C09089=1078.091,60.474,-64.485,173.827,22.395,153.881
C09090=1078.085,60.225,-64.469,173.826,22.393,153.880
C09091=1078.079,59.976,-64.451,173.824,22.391,153.880
C09092=1078.073,59.726,-64.435,173.822,22.388,153.880
C09093=1078.067,59.477,-64.419,173.821,22.386,153.880
C09094=1078.061,59.228,-64.403,173.820,22.383,153.879
C09095=1078.056,58.978,-64.386,173.818,22.381,153.879
C09096=1078.050,58.729,-64.369,173.816,22.379,153.879
C09097=1078.044,58.480,-64.352,173.815,22.376,153.879
C09098=1078.038,58.230,-64.336,173.814,22.374,153.878
C09099=1078.033,57.981,-64.319,173.812,22.371,153.878
C09100=1078.027,57.731,-64.303,173.810,22.369,153.878
C09101=1078.021,57.482,-64.287,173.809,22.367,153.878
C09102=1078.015,57.233,-64.271,173.807,22.364,153.877
C09103=1078.010,56.983,-64.254,173.806,22.362,153.877
C09104=1078.004,56.734,-64.237,173.804,22.359,153.877
C09105=1077.998,56.484,-64.221,173.803,22.357,153.877
C09106=1077.992,56.235,-64.205,173.801,22.354,153.876
C09107=1077.986,55.986,-64.189,173.800,22.352,153.876
C09108=1077.981,55.736,-64.172,173.798,22.350,153.876
C09109=1077.975,55.487,-64.156,173.796,22.347,153.876
C09110=1077.969,55.237,-64.139,173.795,22.344,153.875
C09111=1077.963,54.988,-64.123,173.794,22.342,153.875
C09112=1077.957,54.739,-64.107,173.793,22.340,153.875
C09113=1077.952,54.489,-64.090,173.790,22.337,153.875
C09114=1077.946,54.240,-64.074,173.789,22.335,153.874
C09115=1077.940,53.990,-64.057,173.788,22.332,153.874
C09116=1077.934,53.741,-64.041,173.787,22.330,153.874
C09117=1077.928,53.492,-64.025,173.785,22.328,153.874
C09118=1077.923,53.242,-64.008,173.783,22.325,153.873
C09119=1077.917,52.993,-63.992,173.782,22.323,153.873
C09120=1077.911,52.743,-63.976,173.780,22.320,153.873
C09121=1077.905,52.494,-63.959,173.779,22.317,153.872
C09122=1077.899,52.245,-63.943,173.777,22.316,153.872
C09123=1077.893,51.995,-63.927,173.776,22.313,153.872
C09124=1077.887,51.746,-63.911,173.774,22.310,153.872
C09125=1077.882,51.496,-63.894,173.773,22.308,153.871
C09126=1077.876,51.246,-63.878,173.772,22.305,153.871
C09127=1077.871,50.998,-63.862,173.770,22.303,153.871
C09128=1077.865,50.748,-63.846,173.768,22.301,153.871
C09129=1077.859,50.499,-63.830,173.767,22.298,153.870
C09130=1077.853,50.250,-63.814,173.766,22.296,153.870
C09131=1077.847,50.000,-63.797,173.764,22.293,153.870
C09132=1077.842,49.751,-63.780,173.762,22.290,153.870
C09133=1077.836,49.501,-63.765,173.761,22.288,153.869
C09134=1077.830,49.251,-63.749,173.760,22.286,153.869
C09135=1077.824,49.002,-63.732,173.758,22.283,153.869
C09136=1077.819,48.753,-63.716,173.757,22.281,153.869
C09137=1077.813,48.504,-63.700,173.755,22.278,153.868
C09138=1077.807,48.254,-63.685,173.754,22.276,153.868
C09139=1077.801,48.005,-63.668,173.752,22.273,153.868
C09140=1077.796,47.755,-63.652,173.751,22.271,153.867
C09141=1077.790,47.506,-63.635,173.750,22.268,153.867
C09142=1077.783,47.225,-63.618,173.747,22.265,153.867
C09143=1077.777,46.944,-63.600,173.746,22.263,153.867
C09144=1077.771,46.663,-63.581,173.744,22.260,153.866
C09145=1077.764,46.383,-63.563,173.743,22.257,153.866
C09146=1077.758,46.133,-63.548,173.741,22.254,153.866
C09147=1077.753,45.883,-63.531,173.740,22.252,153.865
C09148=1077.748,45.635,-63.515,173.738,22.250,153.865
C09149=1077.742,45.385,-63.499,173.737,22.247,153.865
C09150=1077.736,45.135,-63.483,173.735,22.244,153.865
C09151=1077.730,44.886,-63.467,173.734,22.242,153.864
C09152=1077.724,44.637,-63.451,173.733,22.240,153.864
C09153=1077.719,44.387,-63.436,173.732,22.237,153.864
C09154=1077.713,44.138,-63.419,173.729,22.234,153.863
C09155=1077.707,43.889,-63.403,173.728,22.232,153.863
C09156=1077.702,43.639,-63.388,173.727,22.229,153.863
C09157=1077.696,43.389,-63.371,173.726,22.227,153.863
C09158=1077.691,43.140,-63.356,173.724,22.225,153.862
C09159=1077.685,42.891,-63.340,173.722,22.222,153.862
C09160=1077.679,42.641,-63.324,173.721,22.220,153.862
C09161=1077.672,42.392,-63.309,173.720,22.217,153.862
C09162=1077.666,42.142,-63.292,173.718,22.215,153.861
C09163=1077.661,41.893,-63.277,173.716,22.212,153.861
C09164=1077.655,41.644,-63.261,173.715,22.210,153.861
C09165=1077.650,41.394,-63.245,173.714,22.208,153.861
C09166=1077.644,41.144,-63.229,173.712,22.205,153.860
C09167=1077.638,40.895,-63.213,173.711,22.202,153.860
C09168=1077.633,40.646,-63.198,173.709,22.200,153.860
C09169=1077.626,40.397,-63.182,173.708,22.198,153.860
C09170=1077.621,40.147,-63.167,173.706,22.195,153.859
C09171=1077.615,39.897,-63.150,173.705,22.193,153.859
C09172=1077.609,39.647,-63.135,173.704,22.190,153.859
C09173=1077.604,39.399,-63.119,173.702,22.188,153.858
C09174=1077.598,39.149,-63.103,173.700,22.185,153.858
C09175=1077.591,38.900,-63.088,173.699,22.183,153.858
C09176=1077.586,38.650,-63.072,173.698,22.180,153.858
C09177=1077.580,38.401,-63.056,173.697,22.178,153.857
C09178=1077.575,38.151,-63.041,173.694,22.175,153.857
C09179=1077.569,37.902,-63.024,173.693,22.173,153.857
C09180=1077.562,37.652,-63.010,173.692,22.170,153.857
C09181=1077.557,37.404,-62.994,173.691,22.168,153.856
C09182=1077.551,37.154,-62.978,173.689,22.165,153.856
C09183=1077.546,36.904,-62.963,173.687,22.163,153.856
C09184=1077.539,36.655,-62.947,173.686,22.161,153.856
C09185=1077.534,36.405,-62.932,173.685,22.158,153.855
C09186=1077.528,36.156,-62.915,173.683,22.156,153.855
C09187=1077.522,35.906,-62.900,173.681,22.153,153.855
C09188=1077.516,35.656,-62.885,173.680,22.151,153.855
C09189=1077.511,35.408,-62.869,173.679,22.148,153.854
C09190=1077.504,35.158,-62.854,173.678,22.146,153.854
C09191=1077.498,34.909,-62.838,173.676,22.144,153.854
C09192=1077.493,34.659,-62.822,173.674,22.141,153.854
C09193=1077.487,34.410,-62.808,173.673,22.139,153.853
C09194=1077.481,34.160,-62.791,173.672,22.136,153.853
C09195=1077.475,33.911,-62.777,173.670,22.133,153.853
C09196=1077.469,33.662,-62.761,173.669,22.131,153.852
C09197=1077.464,33.412,-62.745,173.667,22.129,153.852
C09198=1077.457,33.163,-62.730,173.666,22.127,153.852
C09199=1077.451,32.913,-62.715,173.664,22.124,153.852
C09200=1077.446,32.664,-62.699,173.663,22.121,153.851
C09201=1077.440,32.414,-62.684,173.661,22.119,153.851
C09202=1077.434,32.164,-62.668,173.660,22.117,153.851
C09203=1077.429,31.915,-62.653,173.659,22.114,153.851
C09204=1077.422,31.666,-62.637,173.657,22.112,153.850
C09205=1077.417,31.416,-62.622,173.656,22.109,153.850
C09206=1077.410,31.135,-62.605,173.655,22.107,153.850
C09207=1077.404,30.854,-62.588,173.653,22.104,153.849
C09208=1077.397,30.574,-62.571,173.651,22.101,153.849
C09209=1077.390,30.293,-62.553,173.649,22.098,153.849
C09210=1077.385,30.043,-62.537,173.648,22.096,153.849
C09211=1077.379,29.795,-62.523,173.647,22.094,153.848
C09212=1077.373,29.545,-62.507,173.645,22.091,153.848
C09213=1077.368,29.296,-62.493,173.644,22.088,153.848
C09214=1077.362,29.046,-62.476,173.642,22.086,153.848
C09215=1077.356,28.796,-62.461,173.641,22.084,153.847
C09216=1077.350,28.547,-62.446,173.639,22.081,153.847
C09217=1077.345,28.297,-62.431,173.638,22.079,153.847
C09218=1077.338,28.048,-62.416,173.637,22.076,153.847
C09219=1077.333,27.798,-62.401,173.635,22.074,153.846
C09220=1077.326,27.549,-62.385,173.634,22.072,153.846
C09221=1077.320,27.300,-62.370,173.632,22.069,153.846
C09222=1077.315,27.050,-62.355,173.631,22.066,153.845
C09223=1077.309,26.801,-62.340,173.629,22.064,153.845
C09224=1077.303,26.551,-62.324,173.628,22.061,153.845
C09225=1077.297,26.302,-62.310,173.626,22.059,153.845
C09226=1077.292,26.052,-62.294,173.625,22.057,153.844
C09227=1077.286,25.803,-62.280,173.624,22.054,153.844
C09228=1077.279,25.553,-62.265,173.622,22.052,153.844
C09229=1077.274,25.303,-62.249,173.621,22.050,153.844
C09230=1077.268,25.054,-62.235,173.619,22.047,153.843
C09231=1077.262,24.804,-62.219,173.618,22.044,153.843
C09232=1077.257,24.555,-62.205,173.617,22.042,153.843
C09233=1077.250,24.306,-62.190,173.615,22.040,153.843
C09234=1077.244,24.056,-62.173,173.614,22.038,153.842
C09235=1077.238,23.807,-62.159,173.612,22.035,153.842
C09236=1077.233,23.558,-62.143,173.611,22.032,153.842
C09237=1077.227,23.309,-62.129,173.610,22.030,153.842
C09238=1077.221,23.059,-62.114,173.608,22.027,153.841
C09239=1077.215,22.809,-62.098,173.607,22.025,153.841
C09240=1077.210,22.559,-62.084,173.605,22.023,153.841
C09241=1077.204,22.309,-62.069,173.604,22.020,153.841
C09242=1077.198,22.060,-62.054,173.602,22.018,153.840
C09243=1077.192,21.811,-62.039,173.601,22.015,153.840
C09244=1077.187,21.562,-62.024,173.599,22.013,153.840
C09245=1077.180,21.312,-62.009,173.598,22.010,153.840
C09246=1077.174,21.063,-61.994,173.597,22.008,153.839
C09247=1077.169,20.813,-61.979,173.595,22.005,153.839
C09248=1077.163,20.564,-61.964,173.594,22.003,153.839
C09249=1077.157,20.314,-61.949,173.592,22.001,153.839
C09250=1077.151,20.064,-61.934,173.591,21.998,153.838
C09251=1077.145,19.815,-61.919,173.590,21.996,153.838
C09252=1077.139,19.566,-61.904,173.588,21.993,153.838
C09253=1077.133,19.316,-61.890,173.587,21.991,153.838
C09254=1077.128,19.066,-61.875,173.585,21.988,153.837
C09255=1077.122,18.817,-61.860,173.584,21.986,153.837
C09256=1077.116,18.568,-61.845,173.583,21.984,153.837
C09257=1077.110,18.319,-61.831,173.581,21.982,153.837
C09258=1077.104,18.069,-61.815,173.580,21.979,153.836
C09259=1077.098,17.820,-61.801,173.578,21.976,153.836
C09260=1077.092,17.569,-61.787,173.577,21.974,153.836
C09261=1077.087,17.320,-61.772,173.576,21.971,153.835
C09262=1077.081,17.070,-61.756,173.574,21.969,153.835
C09263=1077.075,16.822,-61.742,173.573,21.967,153.835
C09264=1077.069,16.572,-61.727,173.571,21.964,153.835
C09265=1077.063,16.322,-61.713,173.570,21.962,153.834
C09266=1077.057,16.073,-61.698,173.568,21.960,153.834
C09267=1077.052,15.823,-61.683,173.567,21.957,153.834
C09268=1077.045,15.574,-61.668,173.566,21.955,153.834
C09269=1077.040,15.324,-61.654,173.564,21.952,153.833
C09270=1077.033,15.045,-61.637,173.563,21.949,153.833
C09271=1077.026,14.765,-61.621,173.561,21.947,153.833
C09272=1077.020,14.486,-61.604,173.560,21.944,153.833
C09273=1077.014,14.207,-61.588,173.558,21.942,153.832
C09274=1077.008,13.957,-61.573,173.556,21.939,153.832
C09275=1077.002,13.708,-61.559,173.555,21.937,153.832
C09276=1076.996,13.458,-61.544,173.554,21.934,153.832
C09277=1076.990,13.209,-61.530,173.553,21.932,153.831
C09278=1076.984,12.959,-61.515,173.551,21.930,153.831
C09279=1076.978,12.710,-61.501,173.549,21.927,153.831
C09280=1076.972,12.460,-61.486,173.548,21.925,153.831
C09281=1076.966,12.211,-61.471,173.547,21.922,153.830
C09282=1076.960,11.961,-61.457,173.545,21.920,153.830
C09283=1076.954,11.712,-61.443,173.544,21.918,153.830
C09284=1076.948,11.462,-61.428,173.542,21.915,153.830
C09285=1076.942,11.213,-61.414,173.541,21.913,153.829
C09286=1076.936,10.963,-61.399,173.539,21.910,153.829
C09287=1076.931,10.713,-61.385,173.538,21.908,153.829
C09288=1076.924,10.464,-61.370,173.537,21.906,153.829
C09289=1076.918,10.215,-61.355,173.535,21.903,153.828
C09290=1076.913,9.965,-61.342,173.534,21.901,153.828
C09291=1076.906,9.715,-61.327,173.532,21.899,153.828
C09292=1076.901,9.466,-61.313,173.531,21.896,153.828
C09293=1076.895,9.216,-61.298,173.530,21.894,153.827
C09294=1076.889,8.967,-61.283,173.529,21.892,153.827
C09295=1076.882,8.717,-61.270,173.526,21.889,153.827
C09296=1076.876,8.468,-61.255,173.525,21.887,153.827
C09297=1076.871,8.219,-61.241,173.524,21.884,153.826
C09298=1076.864,7.969,-61.226,173.523,21.882,153.826
C09299=1076.859,7.720,-61.212,173.522,21.880,153.826
C09300=1076.853,7.470,-61.197,173.520,21.877,153.826
C09301=1076.847,7.220,-61.184,173.518,21.875,153.825
C09302=1076.841,6.971,-61.169,173.517,21.872,153.825
C09303=1076.835,6.721,-61.155,173.516,21.870,153.825
C09304=1076.829,6.472,-61.140,173.514,21.868,153.825
C09305=1076.823,6.222,-61.126,173.512,21.865,153.824
C09306=1076.818,5.973,-61.111,173.511,21.863,153.824
C09307=1076.812,5.723,-61.097,173.510,21.860,153.824
C09308=1076.806,5.473,-61.083,173.509,21.858,153.824
C09309=1076.800,5.224,-61.069,173.507,21.856,153.823
C09310=1076.795,4.975,-61.055,173.506,21.853,153.823
C09311=1076.788,4.725,-61.040,173.504,21.851,153.823
C09312=1076.782,4.476,-61.027,173.503,21.848,153.823
C09313=1076.776,4.227,-61.012,173.502,21.846,153.822
C09314=1076.770,3.976,-60.998,173.500,21.844,153.822
C09315=1076.765,3.727,-60.984,173.499,21.842,153.822
C09316=1076.759,3.478,-60.969,173.497,21.839,153.822
C09317=1076.753,3.228,-60.955,173.496,21.836,153.821
C09318=1076.747,2.979,-60.940,173.494,21.834,153.821
C09319=1076.742,2.729,-60.927,173.493,21.832,153.821
C09320=1076.736,2.479,-60.912,173.492,21.829,153.821
C09321=1076.730,2.230,-60.898,173.491,21.827,153.820
C09322=1076.724,1.981,-60.885,173.489,21.825,153.820
C09323=1076.718,1.731,-60.871,173.488,21.822,153.820
C09324=1076.712,1.481,-60.856,173.486,21.820,153.820
C09325=1076.706,1.232,-60.842,173.485,21.818,153.819
C09326=1076.701,0.982,-60.828,173.484,21.815,153.819
C09327=1076.694,0.733,-60.813,173.483,21.813,153.819
C09328=1076.689,0.483,-60.799,173.480,21.810,153.819
C09329=1076.683,0.233,-60.785,173.479,21.808,153.818
C09330=1076.677,-0.016,-60.772,173.478,21.805,153.818
C09331=1076.671,-0.266,-60.757,173.477,21.803,153.818
C09332=1076.665,-0.515,-60.743,173.475,21.801,153.818
C09333=1076.660,-0.765,-60.729,173.473,21.798,153.817
C09334=1076.655,-0.977,-60.717,173.473,21.797,153.817
C09335=1076.650,-1.191,-60.706,173.472,21.795,153.817
C09336=1076.645,-1.403,-60.693,173.470,21.792,153.817
C09337=1076.640,-1.617,-60.681,173.469,21.790,153.817
C09338=1076.635,-1.828,-60.670,173.468,21.788,153.816
C09339=1076.630,-2.042,-60.658,173.466,21.786,153.816
C09340=1076.625,-2.255,-60.645,173.465,21.784,153.816
C09341=1076.620,-2.468,-60.634,173.465,21.782,153.816
C09342=1076.615,-2.717,-60.620,173.463,21.780,153.816
C09343=1076.609,-2.966,-60.605,173.461,21.777,153.815
C09344=1076.603,-3.216,-60.591,173.460,21.775,153.815
C09345=1076.597,-3.466,-60.577,173.459,21.773,153.815
C09346=1076.591,-3.715,-60.564,173.458,21.770,153.814
C09347=1076.586,-3.965,-60.550,173.456,21.768,153.814
C09348=1076.579,-4.215,-60.537,173.454,21.765,153.814
C09349=1076.573,-4.464,-60.522,173.453,21.763,153.814
C09350=1076.567,-4.713,-60.508,173.452,21.761,153.814
C09351=1076.561,-4.963,-60.495,173.450,21.759,153.813
C09352=1076.555,-5.213,-60.481,173.449,21.757,153.813
C09353=1076.549,-5.462,-60.467,173.448,21.754,153.813
C09354=1076.543,-5.712,-60.454,173.446,21.752,153.813
C09355=1076.538,-5.961,-60.440,173.445,21.749,153.812
C09356=1076.531,-6.211,-60.426,173.443,21.747,153.812
C09357=1076.526,-6.461,-60.412,173.442,21.745,153.812
C09358=1076.517,-6.811,-60.392,173.440,21.742,153.812
C09359=1076.509,-7.162,-60.373,173.438,21.738,153.811
C09360=1076.501,-7.513,-60.354,173.436,21.735,153.811
C09361=1076.492,-7.863,-60.334,173.434,21.732,153.811
C09362=1076.486,-8.113,-60.321,173.433,21.730,153.810
C09363=1076.480,-8.362,-60.307,173.431,21.727,153.810
C09364=1076.475,-8.612,-60.293,173.430,21.725,153.810
C09365=1076.468,-8.862,-60.280,173.428,21.722,153.810
C09366=1076.462,-9.111,-60.266,173.427,21.720,153.810
C09367=1076.456,-9.361,-60.253,173.426,21.718,153.809
C09368=1076.451,-9.610,-60.239,173.425,21.716,153.809
C09369=1076.444,-9.859,-60.226,173.422,21.713,153.809
C09370=1076.439,-10.109,-60.212,173.421,21.711,153.809
C09371=1076.432,-10.359,-60.198,173.420,21.709,153.808
C09372=1076.427,-10.609,-60.184,173.419,21.707,153.808
C09373=1076.422,-10.859,-60.171,173.417,21.704,153.808
C09374=1076.415,-11.108,-60.158,173.416,21.702,153.808
C09375=1076.410,-11.358,-60.144,173.414,21.699,153.808
C09376=1076.404,-11.607,-60.131,173.413,21.697,153.807
C09377=1076.398,-11.856,-60.117,173.411,21.695,153.807
C09378=1076.391,-12.106,-60.103,173.410,21.692,153.807
C09379=1076.386,-12.356,-60.089,173.409,21.691,153.807
C09380=1076.380,-12.605,-60.076,173.408,21.688,153.806
C09381=1076.374,-12.855,-60.062,173.405,21.686,153.806
C09382=1076.368,-13.104,-60.049,173.404,21.683,153.806
C09383=1076.362,-13.354,-60.035,173.403,21.681,153.806
C09384=1076.357,-13.603,-60.022,173.402,21.679,153.806
C09385=1076.351,-13.853,-60.009,173.401,21.676,153.805
C09386=1076.345,-14.102,-59.995,173.399,21.674,153.805
C09387=1076.339,-14.352,-59.981,173.398,21.672,153.805
C09388=1076.333,-14.602,-59.968,173.396,21.670,153.805
C09389=1076.327,-14.851,-59.954,173.395,21.667,153.804
C09390=1076.321,-15.101,-59.941,173.393,21.665,153.804
C09391=1076.315,-15.351,-59.928,173.392,21.663,153.804
C09392=1076.310,-15.600,-59.914,173.391,21.661,153.804
C09393=1076.303,-15.849,-59.901,173.390,21.658,153.803
C09394=1076.297,-16.099,-59.888,173.387,21.656,153.803
C09395=1076.292,-16.348,-59.874,173.386,21.653,153.803
C09396=1076.286,-16.598,-59.861,173.385,21.651,153.803
C09397=1076.279,-16.848,-59.848,173.384,21.649,153.803
C09398=1076.273,-17.123,-59.833,173.382,21.647,153.802
C09399=1076.266,-17.400,-59.818,173.380,21.644,153.802
C09400=1076.260,-17.675,-59.803,173.379,21.642,153.802
C09401=1076.253,-17.951,-59.789,173.377,21.639,153.802
C09402=1076.247,-18.200,-59.776,173.376,21.637,153.802
C09403=1076.241,-18.450,-59.762,173.374,21.635,153.801
C09404=1076.235,-18.700,-59.749,173.373,21.632,153.801
C09405=1076.229,-18.949,-59.736,173.372,21.630,153.801
C09406=1076.223,-19.198,-59.723,173.370,21.628,153.801
C09407=1076.218,-19.448,-59.710,173.369,21.626,153.800
C09408=1076.211,-19.698,-59.696,173.367,21.624,153.800
C09409=1076.205,-19.948,-59.683,173.366,21.621,153.800
C09410=1076.200,-20.198,-59.669,173.365,21.619,153.800
C09411=1076.193,-20.447,-59.656,173.363,21.617,153.800
C09412=1076.187,-20.696,-59.643,173.362,21.615,153.799
C09413=1076.181,-20.946,-59.630,173.361,21.613,153.799
C09414=1076.176,-21.196,-59.617,173.359,21.610,153.799
C09415=1076.170,-21.445,-59.603,173.357,21.608,153.799
C09416=1076.164,-21.695,-59.591,173.356,21.605,153.799
C09417=1076.157,-21.944,-59.577,173.355,21.604,153.798
C09418=1076.152,-22.194,-59.564,173.354,21.601,153.798
C09419=1076.146,-22.444,-59.551,173.352,21.599,153.798
C09420=1076.140,-22.693,-59.538,173.351,21.597,153.798
C09421=1076.134,-22.943,-59.525,173.350,21.595,153.797
C09422=1076.128,-23.192,-59.512,173.347,21.592,153.797
C09423=1076.122,-23.442,-59.498,173.346,21.590,153.797
C09424=1076.116,-23.692,-59.486,173.345,21.588,153.797
C09425=1076.110,-23.941,-59.472,173.344,21.586,153.797
C09426=1076.104,-24.191,-59.460,173.342,21.583,153.796
C09427=1076.099,-24.440,-59.446,173.341,21.581,153.796
C09428=1076.093,-24.690,-59.433,173.340,21.579,153.796
C09429=1076.087,-24.939,-59.420,173.338,21.577,153.796
C09430=1076.081,-25.189,-59.407,173.336,21.574,153.796
C09431=1076.074,-25.439,-59.394,173.335,21.572,153.795
C09432=1076.070,-25.688,-59.381,173.334,21.570,153.795
C09433=1076.064,-25.937,-59.368,173.333,21.568,153.795
C09434=1076.058,-26.187,-59.356,173.331,21.566,153.795
C09435=1076.052,-26.436,-59.342,173.330,21.563,153.795
C09436=1076.046,-26.686,-59.330,173.328,21.561,153.794
C09437=1076.040,-26.936,-59.316,173.326,21.559,153.794
C09438=1076.034,-27.186,-59.303,173.325,21.557,153.794
C09439=1076.028,-27.435,-59.290,173.324,21.555,153.794
C09440=1076.022,-27.685,-59.278,173.323,21.553,153.794
C09441=1076.016,-27.934,-59.264,173.321,21.551,153.793
C09442=1076.010,-28.184,-59.252,173.320,21.548,153.793
C09443=1076.004,-28.434,-59.239,173.318,21.546,153.793
C09444=1075.998,-28.683,-59.226,173.316,21.544,153.793
C09445=1075.992,-28.933,-59.213,173.315,21.541,153.793
C09446=1075.986,-29.182,-59.200,173.314,21.539,153.792
C09447=1075.980,-29.432,-59.187,173.313,21.537,153.792
C09448=1075.974,-29.682,-59.174,173.311,21.536,153.792
C09449=1075.968,-29.931,-59.162,173.310,21.533,153.792
C09450=1075.962,-30.181,-59.149,173.309,21.531,153.792
C09451=1075.956,-30.431,-59.136,173.306,21.529,153.792
C09452=1075.950,-30.680,-59.123,173.305,21.527,153.791
C09453=1075.944,-30.930,-59.111,173.304,21.524,153.791
C09454=1075.938,-31.179,-59.098,173.303,21.522,153.791
C09455=1075.932,-31.429,-59.085,173.301,21.520,153.791
C09456=1075.926,-31.679,-59.073,173.300,21.518,153.791
C09457=1075.920,-31.928,-59.059,173.299,21.516,153.790
C09458=1075.914,-32.178,-59.047,173.296,21.514,153.790
C09459=1075.908,-32.428,-59.034,173.295,21.512,153.790
C09460=1075.901,-32.677,-59.022,173.294,21.509,153.790
C09461=1075.896,-32.927,-59.009,173.293,21.507,153.790
C09462=1075.890,-33.201,-58.995,173.291,21.505,153.789
C09463=1075.883,-33.476,-58.981,173.289,21.502,153.789
C09464=1075.876,-33.752,-58.968,173.288,21.500,153.789
C09465=1075.870,-34.027,-58.953,173.287,21.498,153.789
C09466=1075.863,-34.276,-58.941,173.285,21.496,153.789
C09467=1075.858,-34.525,-58.929,173.283,21.494,153.789
C09468=1075.852,-34.775,-58.915,173.282,21.492,153.788
C09469=1075.846,-35.024,-58.903,173.281,21.489,153.788
C09470=1075.840,-35.274,-58.890,173.279,21.487,153.788
C09471=1075.834,-35.524,-58.878,173.278,21.485,153.788
C09472=1075.828,-35.774,-58.864,173.277,21.483,153.788
C09473=1075.822,-36.023,-58.852,173.275,21.481,153.787
C09474=1075.817,-36.273,-58.840,173.274,21.479,153.787
C09475=1075.811,-36.522,-58.827,173.272,21.476,153.787
C09476=1075.805,-36.772,-58.814,173.270,21.475,153.787
C09477=1075.799,-37.022,-58.802,173.269,21.473,153.787
C09478=1075.793,-37.271,-58.789,173.268,21.470,153.786
C09479=1075.787,-37.520,-58.777,173.267,21.468,153.786
C09480=1075.781,-37.770,-58.764,173.265,21.466,153.786
C09481=1075.775,-38.020,-58.752,173.264,21.464,153.786
C09482=1075.769,-38.270,-58.739,173.263,21.462,153.786
C09483=1075.763,-38.520,-58.727,173.261,21.460,153.786
C09484=1075.758,-38.769,-58.715,173.259,21.457,153.785
C09485=1075.751,-39.018,-58.701,173.258,21.455,153.785
C09486=1075.745,-39.268,-58.689,173.256,21.453,153.785
C09487=1075.739,-39.518,-58.677,173.255,21.452,153.785
C09488=1075.733,-39.768,-58.664,173.254,21.450,153.785
C09489=1075.727,-40.018,-58.652,173.252,21.448,153.785
C09490=1075.721,-40.266,-58.640,173.251,21.446,153.784
C09491=1075.715,-40.516,-58.628,173.250,21.443,153.784
C09492=1075.709,-40.766,-58.615,173.248,21.441,153.784
C09493=1075.703,-41.016,-58.603,173.246,21.439,153.784
C09494=1075.697,-41.266,-58.591,173.245,21.437,153.784
C09495=1075.691,-41.515,-58.578,173.244,21.435,153.784
C09496=1075.685,-41.765,-58.566,173.242,21.433,153.783
C09497=1075.679,-42.014,-58.554,173.241,21.431,153.783
C09498=1075.673,-42.264,-58.541,173.240,21.429,153.783
C09499=1075.667,-42.514,-58.529,173.238,21.427,153.783
C09500=1075.661,-42.762,-58.516,173.237,21.425,153.783
C09501=1075.655,-43.012,-58.504,173.235,21.423,153.783
C09502=1075.649,-43.262,-58.491,173.233,21.421,153.783
C09503=1075.642,-43.512,-58.480,173.232,21.419,153.782
C09504=1075.637,-43.761,-58.468,173.231,21.417,153.782
C09505=1075.631,-44.011,-58.455,173.229,21.414,153.782
C09506=1075.625,-44.261,-58.443,173.228,21.413,153.782
C09507=1075.619,-44.511,-58.431,173.227,21.411,153.782
C09508=1075.613,-44.760,-58.419,173.225,21.409,153.781
C09509=1075.607,-45.010,-58.407,173.224,21.407,153.781
C09510=1075.601,-45.259,-58.394,173.223,21.405,153.781
C09511=1075.595,-45.509,-58.382,173.220,21.402,153.781
C09512=1075.589,-45.758,-58.370,173.219,21.400,153.781
C09513=1075.583,-46.008,-58.357,173.218,21.398,153.781
C09514=1075.577,-46.258,-58.345,173.216,21.396,153.781
C09515=1075.571,-46.507,-58.333,173.215,21.394,153.780
C09516=1075.565,-46.757,-58.321,173.214,21.393,153.780
C09517=1075.559,-47.007,-58.308,173.212,21.391,153.780
C09518=1075.553,-47.256,-58.297,173.211,21.389,153.780
C09519=1075.548,-47.506,-58.285,173.210,21.387,153.780
C09520=1075.542,-47.756,-58.272,173.207,21.384,153.780
C09521=1075.535,-48.005,-58.260,173.206,21.382,153.779
C09522=1075.530,-48.255,-58.248,173.205,21.380,153.779
C09523=1075.523,-48.504,-58.236,173.203,21.378,153.779
C09524=1075.517,-48.754,-58.224,173.202,21.376,153.779
C09525=1075.512,-49.004,-58.212,173.201,21.375,153.779
C09526=1075.505,-49.279,-58.198,173.199,21.373,153.779
C09527=1075.499,-49.555,-58.185,173.197,21.370,153.778
C09528=1075.492,-49.830,-58.171,173.196,21.368,153.778
C09529=1075.486,-50.105,-58.159,173.195,21.366,153.778
C09530=1075.479,-50.355,-58.147,173.193,21.364,153.778
C09531=1075.473,-50.605,-58.134,173.192,21.362,153.778
C09532=1075.467,-50.853,-58.123,173.190,21.359,153.778
C09533=1075.461,-51.103,-58.110,173.188,21.358,153.778
C09534=1075.455,-51.354,-58.099,173.187,21.356,153.778
C09535=1075.449,-51.603,-58.087,173.185,21.354,153.777
C09536=1075.443,-51.852,-58.075,173.184,21.352,153.777
C09537=1075.437,-52.102,-58.063,173.183,21.350,153.777
C09538=1075.430,-52.352,-58.052,173.181,21.348,153.777
C09539=1075.425,-52.601,-58.039,173.180,21.347,153.777
C09540=1075.418,-52.851,-58.028,173.178,21.345,153.777
C09541=1075.412,-53.101,-58.016,173.177,21.343,153.777
C09542=1075.407,-53.350,-58.004,173.176,21.341,153.776
C09543=1075.400,-53.600,-57.992,173.173,21.339,153.776
C09544=1075.393,-53.849,-57.980,173.172,21.337,153.776
C09545=1075.388,-54.100,-57.968,173.171,21.335,153.776
C09546=1075.382,-54.349,-57.957,173.169,21.333,153.776
C09547=1075.375,-54.598,-57.945,173.168,21.331,153.776
C09548=1075.369,-54.849,-57.933,173.167,21.329,153.776
C09549=1075.363,-55.098,-57.921,173.165,21.328,153.776
C09550=1075.357,-55.347,-57.909,173.164,21.326,153.775
C09551=1075.352,-55.597,-57.898,173.162,21.324,153.775
C09552=1075.345,-55.847,-57.886,173.161,21.322,153.775
C09553=1075.339,-56.097,-57.875,173.160,21.320,153.775
C09554=1075.333,-56.346,-57.863,173.158,21.319,153.775
C09555=1075.327,-56.596,-57.851,173.156,21.316,153.775
C09556=1075.320,-56.846,-57.839,173.154,21.314,153.775
C09557=1075.314,-57.095,-57.828,173.153,21.312,153.775
C09558=1075.309,-57.345,-57.816,173.152,21.311,153.775
C09559=1075.302,-57.595,-57.804,173.150,21.309,153.774
C09560=1075.296,-57.844,-57.792,173.149,21.307,153.774
C09561=1075.291,-58.094,-57.780,173.148,21.305,153.774
C09562=1075.284,-58.343,-57.769,173.146,21.304,153.774
C09563=1075.278,-58.593,-57.758,173.145,21.302,153.774
C09564=1075.271,-58.843,-57.746,173.143,21.300,153.774
C09565=1075.266,-59.093,-57.734,173.142,21.298,153.774
C09566=1075.260,-59.342,-57.722,173.140,21.296,153.774
C09567=1075.254,-59.592,-57.711,173.139,21.294,153.773
C09568=1075.247,-59.841,-57.699,173.137,21.292,153.773
C09569=1075.242,-60.091,-57.688,173.135,21.290,153.773
C09570=1075.236,-60.341,-57.676,173.134,21.289,153.773
C09571=1075.229,-60.591,-57.665,173.133,21.287,153.773
C09572=1075.223,-60.840,-57.653,173.131,21.285,153.773
C09573=1075.218,-61.090,-57.641,173.130,21.283,153.773
C09574=1075.212,-61.339,-57.630,173.128,21.281,153.773
C09575=1075.205,-61.589,-57.618,173.127,21.279,153.772
C09576=1075.199,-61.838,-57.607,173.126,21.277,153.772
C09577=1075.194,-62.089,-57.595,173.124,21.276,153.772
C09578=1075.188,-62.337,-57.583,173.123,21.274,153.772
C09579=1075.181,-62.588,-57.572,173.121,21.272,153.772
C09580=1075.175,-62.836,-57.561,173.120,21.271,153.772
C09581=1075.170,-63.087,-57.549,173.119,21.269,153.772
C09582=1075.164,-63.336,-57.538,173.117,21.267,153.772
C09583=1075.157,-63.586,-57.526,173.115,21.265,153.772
C09584=1075.152,-63.835,-57.515,173.113,21.263,153.771
C09585=1075.146,-64.085,-57.503,173.112,21.261,153.771
C09586=1075.140,-64.335,-57.492,173.111,21.260,153.771
C09587=1075.134,-64.585,-57.480,173.109,21.258,153.771
C09588=1075.128,-64.834,-57.469,173.108,21.256,153.771
C09589=1075.121,-65.084,-57.458,173.106,21.254,153.771
C09590=1075.115,-65.360,-57.445,173.105,21.252,153.771
C09591=1075.108,-65.637,-57.432,173.103,21.250,153.771
C09592=1075.102,-65.913,-57.419,173.101,21.248,153.771
C09593=1075.095,-66.191,-57.407,173.100,21.246,153.770
C09594=1075.089,-66.440,-57.396,173.098,21.245,153.770
C09595=1075.083,-66.690,-57.383,173.097,21.243,153.770
C09596=1075.077,-66.940,-57.373,173.096,21.241,153.770
C09597=1075.071,-67.190,-57.361,173.094,21.239,153.770
C09598=1075.065,-67.439,-57.350,173.093,21.237,153.770
C09599=1075.059,-67.689,-57.339,173.091,21.236,153.770
C09600=1075.053,-67.938,-57.328,173.090,21.234,153.770
C09601=1075.048,-68.187,-57.315,173.088,21.232,153.770
C09602=1075.041,-68.438,-57.304,173.086,21.230,153.770
C09603=1075.036,-68.687,-57.293,173.085,21.228,153.769
C09604=1075.029,-68.937,-57.282,173.083,21.227,153.769
C09605=1075.023,-69.186,-57.271,173.082,21.225,153.769
C09606=1075.017,-69.436,-57.260,173.081,21.223,153.769
C09607=1075.012,-69.686,-57.248,173.079,21.221,153.769
C09608=1075.006,-69.936,-57.237,173.078,21.219,153.769
C09609=1074.999,-70.185,-57.225,173.076,21.218,153.769
C09610=1074.994,-70.435,-57.214,173.075,21.216,153.769
C09611=1074.988,-70.684,-57.203,173.073,21.215,153.769
C09612=1074.982,-70.934,-57.192,173.072,21.213,153.769
C09613=1074.976,-71.184,-57.181,173.071,21.211,153.768
C09614=1074.970,-71.434,-57.169,173.069,21.209,153.768
C09615=1074.964,-71.683,-57.158,173.068,21.207,153.768
C09616=1074.959,-71.933,-57.147,173.066,21.206,153.768
C09617=1074.952,-72.183,-57.136,173.065,21.204,153.768
C09618=1074.946,-72.432,-57.125,173.063,21.203,153.768
C09619=1074.941,-72.682,-57.114,173.062,21.201,153.768
C09620=1074.934,-72.932,-57.102,173.060,21.199,153.768
C09621=1074.928,-73.181,-57.091,173.059,21.197,153.768
C09622=1074.923,-73.431,-57.079,173.057,21.195,153.768
C09623=1074.917,-73.681,-57.068,173.055,21.193,153.768
C09624=1074.911,-73.931,-57.057,173.054,21.192,153.768
C09625=1074.906,-74.180,-57.046,173.052,21.190,153.767
C09626=1074.899,-74.430,-57.035,173.051,21.189,153.767
C09627=1074.893,-74.680,-57.024,173.050,21.187,153.767
C09628=1074.887,-74.930,-57.013,173.048,21.185,153.767
C09629=1074.880,-75.178,-57.002,173.046,21.184,153.767
C09630=1074.875,-75.428,-56.991,173.045,21.182,153.767
C09631=1074.868,-75.678,-56.980,173.044,21.180,153.767
C09632=1074.862,-75.928,-56.969,173.042,21.178,153.767
C09633=1074.857,-76.177,-56.958,173.041,21.177,153.767
C09634=1074.850,-76.427,-56.947,173.039,21.176,153.767
C09635=1074.845,-76.677,-56.936,173.038,21.174,153.767
C09636=1074.839,-76.926,-56.925,173.036,21.172,153.767
C09637=1074.833,-77.176,-56.914,173.035,21.171,153.767
C09638=1074.827,-77.426,-56.903,173.033,21.169,153.766
C09639=1074.820,-77.676,-56.892,173.032,21.167,153.766
C09640=1074.814,-77.925,-56.882,173.030,21.165,153.766
C09641=1074.808,-78.175,-56.871,173.029,21.164,153.766
C09642=1074.803,-78.424,-56.860,173.027,21.163,153.766
C09643=1074.796,-78.674,-56.849,173.026,21.161,153.766
C09644=1074.790,-78.924,-56.838,173.024,21.159,153.766
C09645=1074.785,-79.173,-56.827,173.023,21.158,153.766
C09646=1074.778,-79.424,-56.816,173.022,21.156,153.766
C09647=1074.772,-79.673,-56.805,173.020,21.154,153.766
C09648=1074.766,-79.922,-56.794,173.018,21.153,153.766
C09649=1074.760,-80.173,-56.783,173.017,21.152,153.766
C09650=1074.754,-80.422,-56.772,173.016,21.150,153.766
C09651=1074.748,-80.671,-56.762,173.014,21.148,153.766
C09652=1074.742,-80.922,-56.751,173.013,21.147,153.766
C09653=1074.736,-81.171,-56.741,173.011,21.145,153.766
C09654=1074.729,-81.450,-56.728,173.009,21.143,153.766
C09655=1074.722,-81.729,-56.716,173.007,21.142,153.765
C09656=1074.715,-82.007,-56.704,173.006,21.140,153.765
C09657=1074.708,-82.287,-56.693,173.004,21.139,153.765
C09658=1074.702,-82.536,-56.682,173.003,21.137,153.765
C09659=1074.695,-82.786,-56.671,173.001,21.135,153.765
C09660=1074.689,-83.036,-56.660,173.000,21.134,153.765
C09661=1074.684,-83.285,-56.650,172.998,21.132,153.765
C09662=1074.677,-83.535,-56.639,172.997,21.131,153.765
C09663=1074.671,-83.784,-56.628,172.995,21.130,153.765
C09664=1074.665,-84.035,-56.618,172.993,21.128,153.765
C09665=1074.659,-84.284,-56.608,172.992,21.126,153.765
C09666=1074.653,-84.534,-56.596,172.991,21.125,153.765
C09667=1074.647,-84.783,-56.585,172.989,21.123,153.765
C09668=1074.640,-85.033,-56.575,172.988,21.122,153.765
C09669=1074.634,-85.283,-56.565,172.986,21.121,153.765
C09670=1074.629,-85.533,-56.554,172.984,21.119,153.765
C09671=1074.622,-85.782,-56.543,172.983,21.118,153.765
C09672=1074.616,-86.032,-56.533,172.981,21.116,153.765
C09673=1074.610,-86.282,-56.521,172.980,21.114,153.765
C09674=1074.604,-86.532,-56.512,172.978,21.113,153.765
C09675=1074.598,-86.781,-56.501,172.977,21.111,153.765
C09676=1074.592,-87.030,-56.491,172.975,21.110,153.765
C09677=1074.585,-87.280,-56.479,172.974,21.109,153.765
C09678=1074.580,-87.531,-56.469,172.972,21.107,153.765
C09679=1074.573,-87.780,-56.459,172.971,21.106,153.765
C09680=1074.568,-88.029,-56.448,172.969,21.104,153.765
C09681=1074.561,-88.279,-56.437,172.968,21.103,153.765
C09682=1074.555,-88.529,-56.427,172.966,21.102,153.765
C09683=1074.549,-88.779,-56.416,172.965,21.100,153.764
C09684=1074.543,-89.028,-56.406,172.963,21.099,153.764
C09685=1074.538,-89.278,-56.396,172.961,21.097,153.764
C09686=1074.531,-89.528,-56.385,172.960,21.096,153.764
C09687=1074.525,-89.777,-56.374,172.959,21.094,153.764
C09688=1074.519,-90.027,-56.364,172.957,21.092,153.764
C09689=1074.513,-90.277,-56.354,172.955,21.091,153.764
C09690=1074.507,-90.526,-56.343,172.954,21.090,153.764
C09691=1074.500,-90.777,-56.333,172.952,21.088,153.764
C09692=1074.495,-91.026,-56.322,172.951,21.087,153.764
C09693=1074.489,-91.276,-56.311,172.949,21.085,153.764
C09694=1074.483,-91.525,-56.302,172.948,21.084,153.764
C09695=1074.477,-91.775,-56.291,172.946,21.083,153.764
C09696=1074.470,-92.024,-56.281,172.945,21.081,153.764
C09697=1074.464,-92.275,-56.270,172.943,21.080,153.764
C09698=1074.459,-92.524,-56.259,172.942,21.078,153.764
C09699=1074.452,-92.774,-56.250,172.940,21.077,153.764
C09700=1074.447,-93.024,-56.239,172.938,21.075,153.764
C09701=1074.440,-93.273,-56.229,172.937,21.074,153.764
C09702=1074.435,-93.523,-56.218,172.935,21.073,153.764
C09703=1074.428,-93.772,-56.208,172.934,21.071,153.764
C09704=1074.422,-94.023,-56.198,172.932,21.070,153.764
C09705=1074.416,-94.272,-56.187,172.931,21.069,153.764
C09706=1074.410,-94.522,-56.177,172.929,21.067,153.764
C09707=1074.404,-94.771,-56.167,172.927,21.066,153.764
C09708=1074.399,-95.022,-56.157,172.926,21.065,153.764
C09709=1074.393,-95.271,-56.146,172.924,21.063,153.764
C09710=1074.387,-95.521,-56.136,172.923,21.062,153.764
C09711=1074.381,-95.770,-56.125,172.921,21.060,153.764
C09712=1074.375,-96.020,-56.116,172.920,21.059,153.764
C09713=1074.368,-96.270,-56.105,172.918,21.057,153.764
C09714=1074.362,-96.520,-56.095,172.917,21.056,153.764
C09715=1074.356,-96.770,-56.084,172.915,21.055,153.764
C09716=1074.350,-97.019,-56.074,172.914,21.053,153.764
C09717=1074.345,-97.269,-56.064,172.912,21.052,153.764
C09718=1074.337,-97.549,-56.053,172.910,21.050,153.764
C09719=1074.331,-97.831,-56.041,172.909,21.049,153.764
C09720=1074.324,-98.112,-56.029,172.907,21.048,153.764
C09721=1074.317,-98.393,-56.018,172.906,21.047,153.764
C09722=1074.311,-98.642,-56.008,172.904,21.045,153.764
C09723=1074.304,-98.893,-55.998,172.903,21.044,153.764
C09724=1074.299,-99.142,-55.987,172.901,21.043,153.764
C09725=1074.292,-99.392,-55.978,172.899,21.042,153.764
C09726=1074.286,-99.641,-55.968,172.898,21.040,153.764
C09727=1074.281,-99.892,-55.957,172.896,21.039,153.764
C09728=1074.274,-100.141,-55.948,172.894,21.038,153.764
C09729=1074.268,-100.391,-55.938,172.893,21.036,153.764
C09730=1074.262,-100.641,-55.927,172.891,21.035,153.764
C09731=1074.256,-100.890,-55.917,172.890,21.034,153.764
C09732=1074.250,-101.140,-55.908,172.888,21.033,153.764
C09733=1074.243,-101.390,-55.898,172.886,21.031,153.764
C09734=1074.237,-101.640,-55.887,172.885,21.030,153.764
C09735=1074.231,-101.889,-55.877,172.883,21.029,153.764
C09736=1074.225,-102.139,-55.868,172.882,21.028,153.764
C09737=1074.219,-102.389,-55.857,172.880,21.026,153.764
C09738=1074.213,-102.638,-55.847,172.879,21.025,153.764
C09739=1074.207,-102.888,-55.838,172.877,21.024,153.764
C09740=1074.201,-103.138,-55.827,172.875,21.022,153.764
C09741=1074.195,-103.388,-55.817,172.875,21.021,153.764
C09742=1074.189,-103.637,-55.808,172.873,21.021,153.764
C09743=1074.182,-103.887,-55.797,172.871,21.019,153.764
C09744=1074.177,-104.137,-55.787,172.870,21.018,153.764
C09745=1074.171,-104.386,-55.778,172.868,21.017,153.764
C09746=1074.165,-104.636,-55.768,172.866,21.015,153.764
C09747=1074.158,-104.885,-55.758,172.865,21.014,153.764
C09748=1074.153,-105.136,-55.748,172.863,21.013,153.764
C09749=1074.146,-105.385,-55.738,172.862,21.012,153.764
C09750=1074.140,-105.635,-55.728,172.860,21.011,153.765
C09751=1074.134,-105.884,-55.718,172.858,21.009,153.765
C09752=1074.128,-106.134,-55.708,172.857,21.008,153.764
C09753=1074.122,-106.384,-55.698,172.855,21.007,153.765
C09754=1074.116,-106.634,-55.689,172.853,21.006,153.765
C09755=1074.110,-106.883,-55.679,172.852,21.005,153.765
C09756=1074.103,-107.133,-55.669,172.850,21.003,153.765
C09757=1074.098,-107.383,-55.659,172.849,21.003,153.765
C09758=1074.092,-107.633,-55.649,172.848,21.001,153.765
C09759=1074.086,-107.883,-55.640,172.846,21.000,153.765
C09760=1074.079,-108.132,-55.629,172.844,20.999,153.765
C09761=1074.073,-108.382,-55.620,172.843,20.998,153.765
C09762=1074.067,-108.631,-55.610,172.841,20.997,153.765
C09763=1074.061,-108.881,-55.601,172.840,20.995,153.765
C09764=1074.054,-109.131,-55.591,172.838,20.995,153.765
C09765=1074.049,-109.381,-55.581,172.836,20.994,153.765
C09766=1074.043,-109.630,-55.571,172.835,20.992,153.765
C09767=1074.036,-109.880,-55.561,172.833,20.991,153.765
C09768=1074.030,-110.130,-55.552,172.831,20.990,153.765
C09769=1074.024,-110.380,-55.542,172.830,20.989,153.765
C09770=1074.018,-110.630,-55.532,172.829,20.988,153.765
C09771=1074.012,-110.879,-55.523,172.827,20.987,153.765
C09772=1074.005,-111.129,-55.513,172.826,20.986,153.765
C09773=1073.999,-111.379,-55.504,172.824,20.985,153.765
C09774=1073.993,-111.628,-55.493,172.822,20.984,153.765
C09775=1073.987,-111.878,-55.484,172.821,20.983,153.766
C09776=1073.981,-112.128,-55.474,172.819,20.982,153.766
C09777=1073.975,-112.378,-55.464,172.817,20.980,153.766
C09778=1073.969,-112.628,-55.455,172.815,20.979,153.766
C09779=1073.963,-112.877,-55.445,172.814,20.978,153.766
C09780=1073.957,-113.127,-55.435,172.812,20.977,153.766
C09781=1073.950,-113.377,-55.426,172.811,20.977,153.766
C09782=1073.944,-113.655,-55.415,172.809,20.975,153.766
C09783=1073.937,-113.934,-55.405,172.807,20.974,153.766
C09784=1073.931,-114.212,-55.394,172.806,20.973,153.766
C09785=1073.923,-114.491,-55.383,172.804,20.972,153.766
C09786=1073.917,-114.740,-55.374,172.802,20.971,153.766
C09787=1073.911,-114.990,-55.364,172.801,20.969,153.766
C09788=1073.905,-115.240,-55.355,172.799,20.969,153.766
C09789=1073.899,-115.490,-55.345,172.797,20.968,153.767
C09790=1073.893,-115.739,-55.336,172.796,20.967,153.766
C09791=1073.887,-115.989,-55.326,172.795,20.966,153.767
C09792=1073.880,-116.239,-55.316,172.793,20.965,153.767
C09793=1073.874,-116.489,-55.307,172.791,20.964,153.767
C09794=1073.868,-116.739,-55.297,172.790,20.963,153.767
C09795=1073.861,-116.988,-55.288,172.788,20.962,153.767
C09796=1073.855,-117.238,-55.279,172.786,20.961,153.767
C09797=1073.849,-117.487,-55.270,172.784,20.959,153.767
C09798=1073.844,-117.737,-55.261,172.783,20.959,153.767
C09799=1073.837,-117.987,-55.251,172.782,20.958,153.767
C09800=1073.831,-118.237,-55.242,172.780,20.957,153.767
C09801=1073.825,-118.487,-55.232,172.779,20.956,153.767
C09802=1073.819,-118.737,-55.222,172.777,20.955,153.767
C09803=1073.813,-118.986,-55.213,172.775,20.954,153.768
C09804=1073.807,-119.236,-55.203,172.773,20.953,153.768
C09805=1073.800,-119.486,-55.194,172.772,20.952,153.768
C09806=1073.795,-119.735,-55.185,172.770,20.951,153.768
C09807=1073.788,-119.984,-55.176,172.768,20.950,153.768
C09808=1073.782,-120.235,-55.167,172.767,20.950,153.768
C09809=1073.776,-120.485,-55.157,172.766,20.949,153.768
C09810=1073.770,-120.735,-55.148,172.764,20.948,153.768
C09811=1073.764,-120.984,-55.138,172.762,20.946,153.768
C09812=1073.757,-121.234,-55.128,172.761,20.946,153.768
C09813=1073.752,-121.483,-55.119,172.759,20.945,153.768
C09814=1073.745,-121.733,-55.111,172.757,20.944,153.769
C09815=1073.739,-121.983,-55.101,172.755,20.943,153.769
C09816=1073.733,-122.233,-55.092,172.754,20.943,153.769
C09817=1073.727,-122.483,-55.082,172.753,20.942,153.769
C09818=1073.720,-122.733,-55.073,172.751,20.940,153.769
C09819=1073.715,-122.982,-55.064,172.749,20.939,153.769
C09820=1073.709,-123.232,-55.055,172.748,20.938,153.769
C09821=1073.702,-123.482,-55.046,172.746,20.938,153.769
C09822=1073.696,-123.731,-55.036,172.744,20.937,153.769
C09823=1073.690,-123.981,-55.027,172.743,20.936,153.769
C09824=1073.685,-124.231,-55.018,172.742,20.935,153.769
C09825=1073.678,-124.481,-55.009,172.740,20.935,153.770
C09826=1073.671,-124.730,-55.000,172.738,20.934,153.770
C09827=1073.665,-124.980,-54.990,172.736,20.933,153.770
C09828=1073.659,-125.230,-54.981,172.735,20.932,153.770
C09829=1073.653,-125.480,-54.972,172.733,20.931,153.770
C09830=1073.647,-125.729,-54.963,172.731,20.930,153.770
C09831=1073.641,-125.979,-54.954,172.730,20.930,153.770
C09832=1073.635,-126.229,-54.945,172.728,20.929,153.770
C09833=1073.628,-126.479,-54.936,172.727,20.928,153.770
C09834=1073.622,-126.728,-54.926,172.725,20.927,153.771
C09835=1073.617,-126.978,-54.918,172.723,20.926,153.771
C09836=1073.610,-127.228,-54.908,172.721,20.925,153.771
C09837=1073.603,-127.477,-54.899,172.720,20.925,153.771
C09838=1073.598,-127.728,-54.890,172.719,20.924,153.771
C09839=1073.591,-127.979,-54.881,172.717,20.923,153.771
C09840=1073.588,-128.230,-54.871,172.715,20.922,153.771
C09841=1073.586,-128.480,-54.860,172.714,20.919,153.771
C09842=1073.586,-128.734,-54.849,172.713,20.916,153.770
C09843=1073.589,-128.987,-54.835,172.713,20.913,153.770
C09844=1073.595,-129.239,-54.821,172.712,20.908,153.769
C09845=1073.602,-129.490,-54.807,172.712,20.902,153.768
C09846=1073.209,-129.511,-54.965,172.667,21.035,153.800
C09847=1073.201,-129.261,-54.979,172.667,21.041,153.801
C09848=1073.196,-129.008,-54.994,172.667,21.045,153.801
C09849=1073.194,-128.756,-55.006,172.668,21.049,153.802
C09850=1073.193,-128.502,-55.018,172.668,21.053,153.803
C09851=1073.194,-128.252,-55.029,172.670,21.055,153.803
C09852=1073.198,-128.001,-55.039,172.671,21.057,153.803
C09853=1073.204,-127.750,-55.048,172.673,21.058,153.803
C09854=1073.210,-127.500,-55.057,172.675,21.058,153.803
C09855=1073.216,-127.250,-55.067,172.676,21.059,153.802
C09856=1073.223,-127.001,-55.076,172.677,21.060,153.802
C09857=1073.229,-126.750,-55.084,172.679,21.061,153.802
C09858=1073.235,-126.500,-55.094,172.681,21.061,153.802
C09859=1073.240,-126.251,-55.103,172.683,21.062,153.802
C09860=1073.247,-126.002,-55.112,172.684,21.063,153.802
C09861=1073.253,-125.751,-55.121,172.686,21.064,153.802
C09862=1073.259,-125.502,-55.131,172.688,21.065,153.802
C09863=1073.265,-125.252,-55.140,172.689,21.065,153.802
C09864=1073.271,-125.002,-55.148,172.690,21.066,153.801
C09865=1073.278,-124.753,-55.158,172.692,21.067,153.801
C09866=1073.284,-124.503,-55.167,172.694,21.068,153.801
C09867=1073.290,-124.253,-55.177,172.696,21.069,153.801
C09868=1073.297,-124.003,-55.185,172.697,21.070,153.801
C09869=1073.303,-123.753,-55.195,172.699,21.071,153.801
C09870=1073.308,-123.504,-55.204,172.700,21.071,153.801
C09871=1073.315,-123.254,-55.213,172.702,21.072,153.801
C09872=1073.321,-123.004,-55.223,172.704,21.073,153.801
C09873=1073.327,-122.754,-55.232,172.705,21.074,153.801
C09874=1073.333,-122.504,-55.241,172.707,21.075,153.801
C09875=1073.339,-122.255,-55.250,172.709,21.076,153.800
C09876=1073.345,-122.006,-55.259,172.710,21.077,153.800
C09877=1073.351,-121.756,-55.269,172.712,21.078,153.800
C09878=1073.357,-121.505,-55.278,172.713,21.078,153.800
C09879=1073.363,-121.256,-55.287,172.715,21.079,153.800
C09880=1073.370,-121.006,-55.296,172.716,21.080,153.800
C09881=1073.376,-120.756,-55.306,172.718,21.081,153.800
C09882=1073.382,-120.507,-55.315,172.720,21.082,153.800
C09883=1073.388,-120.257,-55.325,172.722,21.083,153.800
C09884=1073.394,-120.008,-55.334,172.723,21.084,153.800
C09885=1073.400,-119.757,-55.343,172.725,21.085,153.800
C09886=1073.406,-119.507,-55.353,172.727,21.086,153.799
C09887=1073.413,-119.258,-55.362,172.728,21.087,153.799
C09888=1073.419,-119.008,-55.372,172.729,21.087,153.799
C09889=1073.425,-118.759,-55.380,172.731,21.088,153.799
C09890=1073.431,-118.509,-55.390,172.733,21.090,153.799
C09891=1073.437,-118.259,-55.400,172.734,21.091,153.799
C09892=1073.444,-118.010,-55.409,172.736,21.091,153.799
C09893=1073.450,-117.760,-55.419,172.738,21.092,153.799
C09894=1073.456,-117.510,-55.428,172.739,21.094,153.799
C09895=1073.462,-117.260,-55.437,172.741,21.095,153.799
C09896=1073.468,-117.010,-55.447,172.742,21.095,153.799
C09897=1073.474,-116.760,-55.456,172.744,21.096,153.798
C09898=1073.480,-116.510,-55.466,172.745,21.097,153.799
C09899=1073.486,-116.261,-55.475,172.747,21.098,153.798
C09900=1073.492,-116.011,-55.485,172.749,21.099,153.798
C09901=1073.498,-115.762,-55.494,172.750,21.100,153.798
C09902=1073.504,-115.512,-55.504,172.752,21.101,153.798
C09903=1073.511,-115.262,-55.513,172.754,21.102,153.798
C09904=1073.517,-115.012,-55.523,172.756,21.104,153.798
C09905=1073.523,-114.762,-55.532,172.757,21.104,153.798
C09906=1073.529,-114.513,-55.542,172.758,21.105,153.798
C09907=1073.536,-114.234,-55.552,172.761,21.107,153.798
C09908=1073.543,-113.955,-55.563,172.762,21.108,153.798
C09909=1073.550,-113.677,-55.574,172.764,21.109,153.798
C09910=1073.556,-113.398,-55.585,172.766,21.110,153.798
C09911=1073.563,-113.149,-55.594,172.767,21.111,153.798
C09912=1073.569,-112.899,-55.604,172.769,21.112,153.798
C09913=1073.575,-112.649,-55.614,172.771,21.113,153.797
C09914=1073.581,-112.399,-55.623,172.772,21.114,153.797
C09915=1073.587,-112.149,-55.633,172.774,21.115,153.797
C09916=1073.593,-111.900,-55.642,172.775,21.116,153.797
C09917=1073.600,-111.650,-55.652,172.776,21.117,153.797
C09918=1073.606,-111.400,-55.661,172.778,21.119,153.797
C09919=1073.612,-111.150,-55.671,172.780,21.119,153.797
C09920=1073.618,-110.901,-55.681,172.782,21.120,153.797
C09921=1073.624,-110.651,-55.691,172.783,21.122,153.797
C09922=1073.630,-110.401,-55.701,172.785,21.123,153.797
C09923=1073.636,-110.151,-55.711,172.786,21.124,153.797
C09924=1073.642,-109.902,-55.720,172.788,21.125,153.797
C09925=1073.649,-109.652,-55.730,172.790,21.126,153.797
C09926=1073.655,-109.402,-55.739,172.791,21.127,153.797
C09927=1073.661,-109.152,-55.749,172.793,21.129,153.797
C09928=1073.667,-108.903,-55.759,172.795,21.129,153.797
C09929=1073.674,-108.653,-55.769,172.795,21.130,153.797
C09930=1073.680,-108.403,-55.778,172.797,21.131,153.797
C09931=1073.685,-108.153,-55.788,172.799,21.133,153.797
C09932=1073.691,-107.904,-55.798,172.800,21.134,153.797
C09933=1073.698,-107.654,-55.808,172.802,21.135,153.797
C09934=1073.704,-107.405,-55.818,172.804,21.136,153.796
C09935=1073.710,-107.155,-55.827,172.805,21.137,153.796
C09936=1073.716,-106.905,-55.837,172.807,21.139,153.796
C09937=1073.722,-106.655,-55.847,172.809,21.140,153.796
C09938=1073.728,-106.406,-55.857,172.810,21.141,153.796
C09939=1073.734,-106.156,-55.867,172.812,21.142,153.796
C09940=1073.741,-105.906,-55.876,172.813,21.143,153.796
C09941=1073.747,-105.656,-55.886,172.815,21.145,153.796
C09942=1073.753,-105.407,-55.897,172.817,21.146,153.796
C09943=1073.759,-105.157,-55.907,172.817,21.147,153.796
C09944=1073.765,-104.907,-55.916,172.819,21.148,153.796
C09945=1073.771,-104.657,-55.926,172.821,21.149,153.796
C09946=1073.777,-104.408,-55.937,172.822,21.150,153.796
C09947=1073.783,-104.158,-55.946,172.824,21.151,153.796
C09948=1073.789,-103.908,-55.956,172.826,21.153,153.796
C09949=1073.795,-103.659,-55.965,172.827,21.154,153.796
C09950=1073.801,-103.409,-55.976,172.829,21.155,153.796
C09951=1073.807,-103.159,-55.986,172.830,21.156,153.796
C09952=1073.813,-102.909,-55.995,172.832,21.158,153.796
C09953=1073.819,-102.660,-56.006,172.834,21.159,153.796
C09954=1073.825,-102.410,-56.016,172.835,21.160,153.796
C09955=1073.831,-102.160,-56.025,172.837,21.161,153.796
C09956=1073.838,-101.911,-56.036,172.838,21.163,153.796
C09957=1073.843,-101.661,-56.046,172.840,21.164,153.796
C09958=1073.850,-101.411,-56.055,172.842,21.165,153.796
C09959=1073.856,-101.162,-56.066,172.843,21.166,153.796
C09960=1073.861,-100.912,-56.076,172.845,21.168,153.796
C09961=1073.869,-100.662,-56.086,172.847,21.169,153.796
C09962=1073.875,-100.412,-56.096,172.847,21.170,153.796
C09963=1073.880,-100.162,-56.106,172.849,21.171,153.796
C09964=1073.887,-99.913,-56.116,172.850,21.173,153.796
C09965=1073.893,-99.663,-56.126,172.852,21.173,153.796
C09966=1073.899,-99.414,-56.137,172.854,21.175,153.796
C09967=1073.905,-99.164,-56.146,172.855,21.176,153.796
C09968=1073.911,-98.914,-56.156,172.857,21.178,153.796
C09969=1073.917,-98.665,-56.167,172.859,21.179,153.796
C09970=1073.923,-98.414,-56.177,172.860,21.180,153.796
C09971=1073.930,-98.134,-56.188,172.862,21.181,153.796
C09972=1073.937,-97.853,-56.199,172.864,21.183,153.796
C09973=1073.944,-97.571,-56.211,172.866,21.185,153.796
C09974=1073.951,-97.290,-56.223,172.867,21.186,153.796
C09975=1073.956,-97.040,-56.233,172.869,21.187,153.796
C09976=1073.963,-96.790,-56.243,172.870,21.189,153.796
C09977=1073.969,-96.540,-56.254,172.872,21.190,153.796
C09978=1073.975,-96.291,-56.264,172.873,21.192,153.796
C09979=1073.980,-96.041,-56.274,172.875,21.193,153.796
C09980=1073.987,-95.792,-56.284,172.876,21.195,153.796
C09981=1073.992,-95.542,-56.294,172.878,21.195,153.796
C09982=1073.999,-95.292,-56.305,172.880,21.197,153.796
C09983=1074.004,-95.042,-56.315,172.881,21.198,153.796
C09984=1074.011,-94.793,-56.325,172.883,21.200,153.796
C09985=1074.016,-94.543,-56.335,172.884,21.201,153.796
C09986=1074.023,-94.293,-56.346,172.886,21.202,153.796
C09987=1074.029,-94.043,-56.356,172.888,21.204,153.796
C09988=1074.035,-93.794,-56.366,172.889,21.205,153.796
C09989=1074.041,-93.544,-56.377,172.891,21.207,153.796
C09990=1074.046,-93.294,-56.387,172.892,21.208,153.796
C09991=1074.053,-93.045,-56.398,172.894,21.210,153.796
C09992=1074.058,-92.795,-56.408,172.895,21.211,153.796
C09993=1074.065,-92.546,-56.418,172.897,21.212,153.796
C09994=1074.071,-92.296,-56.429,172.898,21.214,153.796
C09995=1074.077,-92.046,-56.439,172.900,21.215,153.796
C09996=1074.083,-91.796,-56.450,172.901,21.217,153.796
//INST
///DATE 2021/06/17 10:54
///ATTR SC,RW,RJ
////FRAME ROBOT
///GROUP1 RB1
NOP
MOVL C00000 V=800.0 PL=0
MOVL C00001 V=800.0 PL=0
MOVL C00002 V=800.0 PL=0
MOVL C00003 V=800.0 PL=0
MOVL C00004 V=800.0 PL=0
MOVL C00005 V=800.0 PL=0
MOVL C00006 V=800.0 PL=0
MOVL C00007 V=800.0 PL=0
MOVL C00008 V=800.0 PL=0
MOVL C00009 V=800.0 PL=0
MOVL C00010 V=800.0 PL=0
MOVL C00011 V=800.0 PL=0
MOVL C00012 V=800.0 PL=0
MOVL C00013 V=800.0 PL=0
MOVL C00014 V=800.0 PL=0
MOVL C00015 V=800.0 PL=0
MOVL C00016 V=800.0 PL=0
MOVL C00017 V=800.0 PL=0
MOVL C00018 V=800.0 PL=0
MOVL C00019 V=800.0 PL=0
MOVL C00020 V=800.0 PL=0
MOVL C00021 V=800.0 PL=0
MOVL C00022 V=800.0 PL=0
MOVL C00023 V=800.0 PL=0
MOVL C00024 V=800.0 PL=0
MOVL C00025 V=800.0 PL=0
MOVL C00026 V=800.0 PL=0
MOVL C00027 V=800.0 PL=0
MOVL C00028 V=800.0 PL=0
MOVL C00029 V=800.0 PL=0
MOVL C00030 V=800.0 PL=0
MOVL C00031 V=800.0 PL=0
MOVL C00032 V=800.0 PL=0
MOVL C00033 V=800.0 PL=0
MOVL C00034 V=800.0 PL=0
MOVL C00035 V=800.0 PL=0
MOVL C00036 V=800.0 PL=0
MOVL C00037 V=800.0 PL=0
MOVL C00038 V=800.0 PL=0
MOVL C00039 V=800.0 PL=0
MOVL C00040 V=800.0 PL=0
MOVL C00041 V=800.0 PL=0
MOVL C00042 V=800.0 PL=0
MOVL C00043 V=800.0 PL=0
MOVL C00044 V=800.0 PL=0
MOVL C00045 V=800.0 PL=0
MOVL C00046 V=800.0 PL=0
MOVL C00047 V=800.0 PL=0
MOVL C00048 V=800.0 PL=0
MOVL C00049 V=800.0 PL=0
MOVL C00050 V=800.0 PL=0
MOVL C00051 V=800.0 PL=0
MOVL C00052 V=800.0 PL=0
MOVL C00053 V=800.0 PL=0
MOVL C00054 V=800.0 PL=0
MOVL C00055 V=800.0 PL=0
MOVL C00056 V=800.0 PL=0
MOVL C00057 V=800.0 PL=0
MOVL C00058 V=800.0 PL=0
MOVL C00059 V=800.0 PL=0
MOVL C00060 V=800.0 PL=0
MOVL C00061 V=800.0 PL=0
MOVL C00062 V=800.0 PL=0
MOVL C00063 V=800.0 PL=0
MOVL C00064 V=800.0 PL=0
MOVL C00065 V=800.0 PL=0
MOVL C00066 V=800.0 PL=0
MOVL C00067 V=800.0 PL=0
MOVL C00068 V=800.0 PL=0
MOVL C00069 V=800.0 PL=0
MOVL C00070 V=800.0 PL=0
MOVL C00071 V=800.0 PL=0
MOVL C00072 V=800.0 PL=0
MOVL C00073 V=800.0 PL=0
MOVL C00074 V=800.0 PL=0
MOVL C00075 V=800.0 PL=0
MOVL C00076 V=800.0 PL=0
MOVL C00077 V=800.0 PL=0
MOVL C00078 V=800.0 PL=0
MOVL C00079 V=800.0 PL=0
MOVL C00080 V=800.0 PL=0
MOVL C00081 V=800.0 PL=0
MOVL C00082 V=800.0 PL=0
MOVL C00083 V=800.0 PL=0
MOVL C00084 V=800.0 PL=0
MOVL C00085 V=800.0 PL=0
MOVL C00086 V=800.0 PL=0
MOVL C00087 V=800.0 PL=0
MOVL C00088 V=800.0 PL=0
MOVL C00089 V=800.0 PL=0
MOVL C00090 V=800.0 PL=0
MOVL C00091 V=800.0 PL=0
MOVL C00092 V=800.0 PL=0
MOVL C00093 V=800.0 PL=0
MOVL C00094 V=800.0 PL=0
MOVL C00095 V=800.0 PL=0
MOVL C00096 V=800.0 PL=0
MOVL C00097 V=800.0 PL=0
MOVL C00098 V=800.0 PL=0
MOVL C00099 V=800.0 PL=0
MOVL C00100 V=800.0 PL=0
MOVL C00101 V=800.0 PL=0
MOVL C00102 V=800.0 PL=0
MOVL C00103 V=800.0 PL=0
MOVL C00104 V=800.0 PL=0
MOVL C00105 V=800.0 PL=0
MOVL C00106 V=800.0 PL=0
MOVL C00107 V=800.0 PL=0
MOVL C00108 V=800.0 PL=0
MOVL C00109 V=800.0 PL=0
MOVL C00110 V=800.0 PL=0
MOVL C00111 V=800.0 PL=0
MOVL C00112 V=800.0 PL=0
MOVL C00113 V=800.0 PL=0
MOVL C00114 V=800.0 PL=0
MOVL C00115 V=800.0 PL=0
MOVL C00116 V=800.0 PL=0
MOVL C00117 V=800.0 PL=0
MOVL C00118 V=800.0 PL=0
MOVL C00119 V=800.0 PL=0
MOVL C00120 V=800.0 PL=0
MOVL C00121 V=800.0 PL=0
MOVL C00122 V=800.0 PL=0
MOVL C00123 V=800.0 PL=0
MOVL C00124 V=800.0 PL=0
MOVL C00125 V=800.0 PL=0
MOVL C00126 V=800.0 PL=0
MOVL C00127 V=800.0 PL=0
MOVL C00128 V=800.0 PL=0
MOVL C00129 V=800.0 PL=0
MOVL C00130 V=800.0 PL=0
MOVL C00131 V=800.0 PL=0
MOVL C00132 V=800.0 PL=0
MOVL C00133 V=800.0 PL=0
MOVL C00134 V=800.0 PL=0
MOVL C00135 V=800.0 PL=0
MOVL C00136 V=800.0 PL=0
MOVL C00137 V=800.0 PL=0
MOVL C00138 V=800.0 PL=0
MOVL C00139 V=800.0 PL=0
MOVL C00140 V=800.0 PL=0
MOVL C00141 V=800.0 PL=0
MOVL C00142 V=800.0 PL=0
MOVL C00143 V=800.0 PL=0
MOVL C00144 V=800.0 PL=0
MOVL C00145 V=800.0 PL=0
MOVL C00146 V=800.0 PL=0
MOVL C00147 V=800.0 PL=0
MOVL C00148 V=800.0 PL=0
MOVL C00149 V=800.0 PL=0
MOVL C00150 V=800.0 PL=0
MOVL C00151 V=800.0 PL=0
MOVL C00152 V=800.0 PL=0
MOVL C00153 V=800.0 PL=0
MOVL C00154 V=800.0 PL=0
MOVL C00155 V=800.0 PL=0
MOVL C00156 V=800.0 PL=0
MOVL C00157 V=800.0 PL=0
MOVL C00158 V=800.0 PL=0
MOVL C00159 V=800.0 PL=0
MOVL C00160 V=800.0 PL=0
MOVL C00161 V=800.0 PL=0
MOVL C00162 V=800.0 PL=0
MOVL C00163 V=800.0 PL=0
MOVL C00164 V=800.0 PL=0
MOVL C00165 V=800.0 PL=0
MOVL C00166 V=800.0 PL=0
MOVL C00167 V=800.0 PL=0
MOVL C00168 V=800.0 PL=0
MOVL C00169 V=800.0 PL=0
MOVL C00170 V=800.0 PL=0
MOVL C00171 V=800.0 PL=0
MOVL C00172 V=800.0 PL=0
MOVL C00173 V=800.0 PL=0
MOVL C00174 V=800.0 PL=0
MOVL C00175 V=800.0 PL=0
MOVL C00176 V=800.0 PL=0
MOVL C00177 V=800.0 PL=0
MOVL C00178 V=800.0 PL=0
MOVL C00179 V=800.0 PL=0
MOVL C00180 V=800.0 PL=0
MOVL C00181 V=800.0 PL=0
MOVL C00182 V=800.0 PL=0
MOVL C00183 V=800.0 PL=0
MOVL C00184 V=800.0 PL=0
MOVL C00185 V=800.0 PL=0
MOVL C00186 V=800.0 PL=0
MOVL C00187 V=800.0 PL=0
MOVL C00188 V=800.0 PL=0
MOVL C00189 V=800.0 PL=0
MOVL C00190 V=800.0 PL=0
MOVL C00191 V=800.0 PL=0
MOVL C00192 V=800.0 PL=0
MOVL C00193 V=800.0 PL=0
MOVL C00194 V=800.0 PL=0
MOVL C00195 V=800.0 PL=0
MOVL C00196 V=800.0 PL=0
MOVL C00197 V=800.0 PL=0
MOVL C00198 V=800.0 PL=0
MOVL C00199 V=800.0 PL=0
MOVL C00200 V=800.0 PL=0
MOVL C00201 V=800.0 PL=0
MOVL C00202 V=800.0 PL=0
MOVL C00203 V=800.0 PL=0
MOVL C00204 V=800.0 PL=0
MOVL C00205 V=800.0 PL=0
MOVL C00206 V=800.0 PL=0
MOVL C00207 V=800.0 PL=0
MOVL C00208 V=800.0 PL=0
MOVL C00209 V=800.0 PL=0
MOVL C00210 V=800.0 PL=0
MOVL C00211 V=800.0 PL=0
MOVL C00212 V=800.0 PL=0
MOVL C00213 V=800.0 PL=0
MOVL C00214 V=800.0 PL=0
MOVL C00215 V=800.0 PL=0
MOVL C00216 V=800.0 PL=0
MOVL C00217 V=800.0 PL=0
MOVL C00218 V=800.0 PL=0
MOVL C00219 V=800.0 PL=0
MOVL C00220 V=800.0 PL=0
MOVL C00221 V=800.0 PL=0
MOVL C00222 V=800.0 PL=0
MOVL C00223 V=800.0 PL=0
MOVL C00224 V=800.0 PL=0
MOVL C00225 V=800.0 PL=0
MOVL C00226 V=800.0 PL=0
MOVL C00227 V=800.0 PL=0
MOVL C00228 V=800.0 PL=0
MOVL C00229 V=800.0 PL=0
MOVL C00230 V=800.0 PL=0
MOVL C00231 V=800.0 PL=0
MOVL C00232 V=800.0 PL=0
MOVL C00233 V=800.0 PL=0
MOVL C00234 V=800.0 PL=0
MOVL C00235 V=800.0 PL=0
MOVL C00236 V=800.0 PL=0
MOVL C00237 V=800.0 PL=0
MOVL C00238 V=800.0 PL=0
MOVL C00239 V=800.0 PL=0
MOVL C00240 V=800.0 PL=0
MOVL C00241 V=800.0 PL=0
MOVL C00242 V=800.0 PL=0
MOVL C00243 V=800.0 PL=0
MOVL C00244 V=800.0 PL=0
MOVL C00245 V=800.0 PL=0
MOVL C00246 V=800.0 PL=0
MOVL C00247 V=800.0 PL=0
MOVL C00248 V=800.0 PL=0
MOVL C00249 V=800.0 PL=0
MOVL C00250 V=800.0 PL=0
MOVL C00251 V=800.0 PL=0
MOVL C00252 V=800.0 PL=0
MOVL C00253 V=800.0 PL=0
MOVL C00254 V=800.0 PL=0
MOVL C00255 V=800.0 PL=0
MOVL C00256 V=800.0 PL=0
MOVL C00257 V=800.0 PL=0
MOVL C00258 V=800.0 PL=0
MOVL C00259 V=800.0 PL=0
MOVL C00260 V=800.0 PL=0
MOVL C00261 V=800.0 PL=0
MOVL C00262 V=800.0 PL=0
MOVL C00263 V=800.0 PL=0
MOVL C00264 V=800.0 PL=0
MOVL C00265 V=800.0 PL=0
MOVL C00266 V=800.0 PL=0
MOVL C00267 V=800.0 PL=0
MOVL C00268 V=800.0 PL=0
MOVL C00269 V=800.0 PL=0
MOVL C00270 V=800.0 PL=0
MOVL C00271 V=800.0 PL=0
MOVL C00272 V=800.0 PL=0
MOVL C00273 V=800.0 PL=0
MOVL C00274 V=800.0 PL=0
MOVL C00275 V=800.0 PL=0
MOVL C00276 V=800.0 PL=0
MOVL C00277 V=800.0 PL=0
MOVL C00278 V=800.0 PL=0
MOVL C00279 V=800.0 PL=0
MOVL C00280 V=800.0 PL=0
MOVL C00281 V=800.0 PL=0
MOVL C00282 V=800.0 PL=0
MOVL C00283 V=800.0 PL=0
MOVL C00284 V=800.0 PL=0
MOVL C00285 V=800.0 PL=0
MOVL C00286 V=800.0 PL=0
MOVL C00287 V=800.0 PL=0
MOVL C00288 V=800.0 PL=0
MOVL C00289 V=800.0 PL=0
MOVL C00290 V=800.0 PL=0
MOVL C00291 V=800.0 PL=0
MOVL C00292 V=800.0 PL=0
MOVL C00293 V=800.0 PL=0
MOVL C00294 V=800.0 PL=0
MOVL C00295 V=800.0 PL=0
MOVL C00296 V=800.0 PL=0
MOVL C00297 V=800.0 PL=0
MOVL C00298 V=800.0 PL=0
MOVL C00299 V=800.0 PL=0
MOVL C00300 V=800.0 PL=0
MOVL C00301 V=800.0 PL=0
MOVL C00302 V=800.0 PL=0
MOVL C00303 V=800.0 PL=0
MOVL C00304 V=800.0 PL=0
MOVL C00305 V=800.0 PL=0
MOVL C00306 V=800.0 PL=0
MOVL C00307 V=800.0 PL=0
MOVL C00308 V=800.0 PL=0
MOVL C00309 V=800.0 PL=0
MOVL C00310 V=800.0 PL=0
MOVL C00311 V=800.0 PL=0
MOVL C00312 V=800.0 PL=0
MOVL C00313 V=800.0 PL=0
MOVL C00314 V=800.0 PL=0
MOVL C00315 V=800.0 PL=0
MOVL C00316 V=800.0 PL=0
MOVL C00317 V=800.0 PL=0
MOVL C00318 V=800.0 PL=0
MOVL C00319 V=800.0 PL=0
MOVL C00320 V=800.0 PL=0
MOVL C00321 V=800.0 PL=0
MOVL C00322 V=800.0 PL=0
MOVL C00323 V=800.0 PL=0
MOVL C00324 V=800.0 PL=0
MOVL C00325 V=800.0 PL=0
MOVL C00326 V=800.0 PL=0
MOVL C00327 V=800.0 PL=0
MOVL C00328 V=800.0 PL=0
MOVL C00329 V=800.0 PL=0
MOVL C00330 V=800.0 PL=0
MOVL C00331 V=800.0 PL=0
MOVL C00332 V=800.0 PL=0
MOVL C00333 V=800.0 PL=0
MOVL C00334 V=800.0 PL=0
MOVL C00335 V=800.0 PL=0
MOVL C00336 V=800.0 PL=0
MOVL C00337 V=800.0 PL=0
MOVL C00338 V=800.0 PL=0
MOVL C00339 V=800.0 PL=0
MOVL C00340 V=800.0 PL=0
MOVL C00341 V=800.0 PL=0
MOVL C00342 V=800.0 PL=0
MOVL C00343 V=800.0 PL=0
MOVL C00344 V=800.0 PL=0
MOVL C00345 V=800.0 PL=0
MOVL C00346 V=800.0 PL=0
MOVL C00347 V=800.0 PL=0
MOVL C00348 V=800.0 PL=0
MOVL C00349 V=800.0 PL=0
MOVL C00350 V=800.0 PL=0
MOVL C00351 V=800.0 PL=0
MOVL C00352 V=800.0 PL=0
MOVL C00353 V=800.0 PL=0
MOVL C00354 V=800.0 PL=0
MOVL C00355 V=800.0 PL=0
MOVL C00356 V=800.0 PL=0
MOVL C00357 V=800.0 PL=0
MOVL C00358 V=800.0 PL=0
MOVL C00359 V=800.0 PL=0
MOVL C00360 V=800.0 PL=0
MOVL C00361 V=800.0 PL=0
MOVL C00362 V=800.0 PL=0
MOVL C00363 V=800.0 PL=0
MOVL C00364 V=800.0 PL=0
MOVL C00365 V=800.0 PL=0
MOVL C00366 V=800.0 PL=0
MOVL C00367 V=800.0 PL=0
MOVL C00368 V=800.0 PL=0
MOVL C00369 V=800.0 PL=0
MOVL C00370 V=800.0 PL=0
MOVL C00371 V=800.0 PL=0
MOVL C00372 V=800.0 PL=0
MOVL C00373 V=800.0 PL=0
MOVL C00374 V=800.0 PL=0
MOVL C00375 V=800.0 PL=0
MOVL C00376 V=800.0 PL=0
MOVL C00377 V=800.0 PL=0
MOVL C00378 V=800.0 PL=0
MOVL C00379 V=800.0 PL=0
MOVL C00380 V=800.0 PL=0
MOVL C00381 V=800.0 PL=0
MOVL C00382 V=800.0 PL=0
MOVL C00383 V=800.0 PL=0
MOVL C00384 V=800.0 PL=0
MOVL C00385 V=800.0 PL=0
MOVL C00386 V=800.0 PL=0
MOVL C00387 V=800.0 PL=0
MOVL C00388 V=800.0 PL=0
MOVL C00389 V=800.0 PL=0
MOVL C00390 V=800.0 PL=0
MOVL C00391 V=800.0 PL=0
MOVL C00392 V=800.0 PL=0
MOVL C00393 V=800.0 PL=0
MOVL C00394 V=800.0 PL=0
MOVL C00395 V=800.0 PL=0
MOVL C00396 V=800.0 PL=0
MOVL C00397 V=800.0 PL=0
MOVL C00398 V=800.0 PL=0
MOVL C00399 V=800.0 PL=0
MOVL C00400 V=800.0 PL=0
MOVL C00401 V=800.0 PL=0
MOVL C00402 V=800.0 PL=0
MOVL C00403 V=800.0 PL=0
MOVL C00404 V=800.0 PL=0
MOVL C00405 V=800.0 PL=0
MOVL C00406 V=800.0 PL=0
MOVL C00407 V=800.0 PL=0
MOVL C00408 V=800.0 PL=0
MOVL C00409 V=800.0 PL=0
MOVL C00410 V=800.0 PL=0
MOVL C00411 V=800.0 PL=0
MOVL C00412 V=800.0 PL=0
MOVL C00413 V=800.0 PL=0
MOVL C00414 V=800.0 PL=0
MOVL C00415 V=800.0 PL=0
MOVL C00416 V=800.0 PL=0
MOVL C00417 V=800.0 PL=0
MOVL C00418 V=800.0 PL=0
MOVL C00419 V=800.0 PL=0
MOVL C00420 V=800.0 PL=0
MOVL C00421 V=800.0 PL=0
MOVL C00422 V=800.0 PL=0
MOVL C00423 V=800.0 PL=0
MOVL C00424 V=800.0 PL=0
MOVL C00425 V=800.0 PL=0
MOVL C00426 V=800.0 PL=0
MOVL C00427 V=800.0 PL=0
MOVL C00428 V=800.0 PL=0
MOVL C00429 V=800.0 PL=0
MOVL C00430 V=800.0 PL=0
MOVL C00431 V=800.0 PL=0
MOVL C00432 V=800.0 PL=0
MOVL C00433 V=800.0 PL=0
MOVL C00434 V=800.0 PL=0
MOVL C00435 V=800.0 PL=0
MOVL C00436 V=800.0 PL=0
MOVL C00437 V=800.0 PL=0
MOVL C00438 V=800.0 PL=0
MOVL C00439 V=800.0 PL=0
MOVL C00440 V=800.0 PL=0
MOVL C00441 V=800.0 PL=0
MOVL C00442 V=800.0 PL=0
MOVL C00443 V=800.0 PL=0
MOVL C00444 V=800.0 PL=0
MOVL C00445 V=800.0 PL=0
MOVL C00446 V=800.0 PL=0
MOVL C00447 V=800.0 PL=0
MOVL C00448 V=800.0 PL=0
MOVL C00449 V=800.0 PL=0
MOVL C00450 V=800.0 PL=0
MOVL C00451 V=800.0 PL=0
MOVL C00452 V=800.0 PL=0
MOVL C00453 V=800.0 PL=0
MOVL C00454 V=800.0 PL=0
MOVL C00455 V=800.0 PL=0
MOVL C00456 V=800.0 PL=0
MOVL C00457 V=800.0 PL=0
MOVL C00458 V=800.0 PL=0
MOVL C00459 V=800.0 PL=0
MOVL C00460 V=800.0 PL=0
MOVL C00461 V=800.0 PL=0
MOVL C00462 V=800.0 PL=0
MOVL C00463 V=800.0 PL=0
MOVL C00464 V=800.0 PL=0
MOVL C00465 V=800.0 PL=0
MOVL C00466 V=800.0 PL=0
MOVL C00467 V=800.0 PL=0
MOVL C00468 V=800.0 PL=0
MOVL C00469 V=800.0 PL=0
MOVL C00470 V=800.0 PL=0
MOVL C00471 V=800.0 PL=0
MOVL C00472 V=800.0 PL=0
MOVL C00473 V=800.0 PL=0
MOVL C00474 V=800.0 PL=0
MOVL C00475 V=800.0 PL=0
MOVL C00476 V=800.0 PL=0
MOVL C00477 V=800.0 PL=0
MOVL C00478 V=800.0 PL=0
MOVL C00479 V=800.0 PL=0
MOVL C00480 V=800.0 PL=0
MOVL C00481 V=800.0 PL=0
MOVL C00482 V=800.0 PL=0
MOVL C00483 V=800.0 PL=0
MOVL C00484 V=800.0 PL=0
MOVL C00485 V=800.0 PL=0
MOVL C00486 V=800.0 PL=0
MOVL C00487 V=800.0 PL=0
MOVL C00488 V=800.0 PL=0
MOVL C00489 V=800.0 PL=0
MOVL C00490 V=800.0 PL=0
MOVL C00491 V=800.0 PL=0
MOVL C00492 V=800.0 PL=0
MOVL C00493 V=800.0 PL=0
MOVL C00494 V=800.0 PL=0
MOVL C00495 V=800.0 PL=0
MOVL C00496 V=800.0 PL=0
MOVL C00497 V=800.0 PL=0
MOVL C00498 V=800.0 PL=0
MOVL C00499 V=800.0 PL=0
MOVL C00500 V=800.0 PL=0
MOVL C00501 V=800.0 PL=0
MOVL C00502 V=800.0 PL=0
MOVL C00503 V=800.0 PL=0
MOVL C00504 V=800.0 PL=0
MOVL C00505 V=800.0 PL=0
MOVL C00506 V=800.0 PL=0
MOVL C00507 V=800.0 PL=0
MOVL C00508 V=800.0 PL=0
MOVL C00509 V=800.0 PL=0
MOVL C00510 V=800.0 PL=0
MOVL C00511 V=800.0 PL=0
MOVL C00512 V=800.0 PL=0
MOVL C00513 V=800.0 PL=0
MOVL C00514 V=800.0 PL=0
MOVL C00515 V=800.0 PL=0
MOVL C00516 V=800.0 PL=0
MOVL C00517 V=800.0 PL=0
MOVL C00518 V=800.0 PL=0
MOVL C00519 V=800.0 PL=0
MOVL C00520 V=800.0 PL=0
MOVL C00521 V=800.0 PL=0
MOVL C00522 V=800.0 PL=0
MOVL C00523 V=800.0 PL=0
MOVL C00524 V=800.0 PL=0
MOVL C00525 V=800.0 PL=0
MOVL C00526 V=800.0 PL=0
MOVL C00527 V=800.0 PL=0
MOVL C00528 V=800.0 PL=0
MOVL C00529 V=800.0 PL=0
MOVL C00530 V=800.0 PL=0
MOVL C00531 V=800.0 PL=0
MOVL C00532 V=800.0 PL=0
MOVL C00533 V=800.0 PL=0
MOVL C00534 V=800.0 PL=0
MOVL C00535 V=800.0 PL=0
MOVL C00536 V=800.0 PL=0
MOVL C00537 V=800.0 PL=0
MOVL C00538 V=800.0 PL=0
MOVL C00539 V=800.0 PL=0
MOVL C00540 V=800.0 PL=0
MOVL C00541 V=800.0 PL=0
MOVL C00542 V=800.0 PL=0
MOVL C00543 V=800.0 PL=0
MOVL C00544 V=800.0 PL=0
MOVL C00545 V=800.0 PL=0
MOVL C00546 V=800.0 PL=0
MOVL C00547 V=800.0 PL=0
MOVL C00548 V=800.0 PL=0
MOVL C00549 V=800.0 PL=0
MOVL C00550 V=800.0 PL=0
MOVL C00551 V=800.0 PL=0
MOVL C00552 V=800.0 PL=0
MOVL C00553 V=800.0 PL=0
MOVL C00554 V=800.0 PL=0
MOVL C00555 V=800.0 PL=0
MOVL C00556 V=800.0 PL=0
MOVL C00557 V=800.0 PL=0
MOVL C00558 V=800.0 PL=0
MOVL C00559 V=800.0 PL=0
MOVL C00560 V=800.0 PL=0
MOVL C00561 V=800.0 PL=0
MOVL C00562 V=800.0 PL=0
MOVL C00563 V=800.0 PL=0
MOVL C00564 V=800.0 PL=0
MOVL C00565 V=800.0 PL=0
MOVL C00566 V=800.0 PL=0
MOVL C00567 V=800.0 PL=0
MOVL C00568 V=800.0 PL=0
MOVL C00569 V=800.0 PL=0
MOVL C00570 V=800.0 PL=0
MOVL C00571 V=800.0 PL=0
MOVL C00572 V=800.0 PL=0
MOVL C00573 V=800.0 PL=0
MOVL C00574 V=800.0 PL=0
MOVL C00575 V=800.0 PL=0
MOVL C00576 V=800.0 PL=0
MOVL C00577 V=800.0 PL=0
MOVL C00578 V=800.0 PL=0
MOVL C00579 V=800.0 PL=0
MOVL C00580 V=800.0 PL=0
MOVL C00581 V=800.0 PL=0
MOVL C00582 V=800.0 PL=0
MOVL C00583 V=800.0 PL=0
MOVL C00584 V=800.0 PL=0
MOVL C00585 V=800.0 PL=0
MOVL C00586 V=800.0 PL=0
MOVL C00587 V=800.0 PL=0
MOVL C00588 V=800.0 PL=0
MOVL C00589 V=800.0 PL=0
MOVL C00590 V=800.0 PL=0
MOVL C00591 V=800.0 PL=0
MOVL C00592 V=800.0 PL=0
MOVL C00593 V=800.0 PL=0
MOVL C00594 V=800.0 PL=0
MOVL C00595 V=800.0 PL=0
MOVL C00596 V=800.0 PL=0
MOVL C00597 V=800.0 PL=0
MOVL C00598 V=800.0 PL=0
MOVL C00599 V=800.0 PL=0
MOVL C00600 V=800.0 PL=0
MOVL C00601 V=800.0 PL=0
MOVL C00602 V=800.0 PL=0
MOVL C00603 V=800.0 PL=0
MOVL C00604 V=800.0 PL=0
MOVL C00605 V=800.0 PL=0
MOVL C00606 V=800.0 PL=0
MOVL C00607 V=800.0 PL=0
MOVL C00608 V=800.0 PL=0
MOVL C00609 V=800.0 PL=0
MOVL C00610 V=800.0 PL=0
MOVL C00611 V=800.0 PL=0
MOVL C00612 V=800.0 PL=0
MOVL C00613 V=800.0 PL=0
MOVL C00614 V=800.0 PL=0
MOVL C00615 V=800.0 PL=0
MOVL C00616 V=800.0 PL=0
MOVL C00617 V=800.0 PL=0
MOVL C00618 V=800.0 PL=0
MOVL C00619 V=800.0 PL=0
MOVL C00620 V=800.0 PL=0
MOVL C00621 V=800.0 PL=0
MOVL C00622 V=800.0 PL=0
MOVL C00623 V=800.0 PL=0
MOVL C00624 V=800.0 PL=0
MOVL C00625 V=800.0 PL=0
MOVL C00626 V=800.0 PL=0
MOVL C00627 V=800.0 PL=0
MOVL C00628 V=800.0 PL=0
MOVL C00629 V=800.0 PL=0
MOVL C00630 V=800.0 PL=0
MOVL C00631 V=800.0 PL=0
MOVL C00632 V=800.0 PL=0
MOVL C00633 V=800.0 PL=0
MOVL C00634 V=800.0 PL=0
MOVL C00635 V=800.0 PL=0
MOVL C00636 V=800.0 PL=0
MOVL C00637 V=800.0 PL=0
MOVL C00638 V=800.0 PL=0
MOVL C00639 V=800.0 PL=0
MOVL C00640 V=800.0 PL=0
MOVL C00641 V=800.0 PL=0
MOVL C00642 V=800.0 PL=0
MOVL C00643 V=800.0 PL=0
MOVL C00644 V=800.0 PL=0
MOVL C00645 V=800.0 PL=0
MOVL C00646 V=800.0 PL=0
MOVL C00647 V=800.0 PL=0
MOVL C00648 V=800.0 PL=0
MOVL C00649 V=800.0 PL=0
MOVL C00650 V=800.0 PL=0
MOVL C00651 V=800.0 PL=0
MOVL C00652 V=800.0 PL=0
MOVL C00653 V=800.0 PL=0
MOVL C00654 V=800.0 PL=0
MOVL C00655 V=800.0 PL=0
MOVL C00656 V=800.0 PL=0
MOVL C00657 V=800.0 PL=0
MOVL C00658 V=800.0 PL=0
MOVL C00659 V=800.0 PL=0
MOVL C00660 V=800.0 PL=0
MOVL C00661 V=800.0 PL=0
MOVL C00662 V=800.0 PL=0
MOVL C00663 V=800.0 PL=0
MOVL C00664 V=800.0 PL=0
MOVL C00665 V=800.0 PL=0
MOVL C00666 V=800.0 PL=0
MOVL C00667 V=800.0 PL=0
MOVL C00668 V=800.0 PL=0
MOVL C00669 V=800.0 PL=0
MOVL C00670 V=800.0 PL=0
MOVL C00671 V=800.0 PL=0
MOVL C00672 V=800.0 PL=0
MOVL C00673 V=800.0 PL=0
MOVL C00674 V=800.0 PL=0
MOVL C00675 V=800.0 PL=0
MOVL C00676 V=800.0 PL=0
MOVL C00677 V=800.0 PL=0
MOVL C00678 V=800.0 PL=0
MOVL C00679 V=800.0 PL=0
MOVL C00680 V=800.0 PL=0
MOVL C00681 V=800.0 PL=0
MOVL C00682 V=800.0 PL=0
MOVL C00683 V=800.0 PL=0
MOVL C00684 V=800.0 PL=0
MOVL C00685 V=800.0 PL=0
MOVL C00686 V=800.0 PL=0
MOVL C00687 V=800.0 PL=0
MOVL C00688 V=800.0 PL=0
MOVL C00689 V=800.0 PL=0
MOVL C00690 V=800.0 PL=0
MOVL C00691 V=800.0 PL=0
MOVL C00692 V=800.0 PL=0
MOVL C00693 V=800.0 PL=0
MOVL C00694 V=800.0 PL=0
MOVL C00695 V=800.0 PL=0
MOVL C00696 V=800.0 PL=0
MOVL C00697 V=800.0 PL=0
MOVL C00698 V=800.0 PL=0
MOVL C00699 V=800.0 PL=0
MOVL C00700 V=800.0 PL=0
MOVL C00701 V=800.0 PL=0
MOVL C00702 V=800.0 PL=0
MOVL C00703 V=800.0 PL=0
MOVL C00704 V=800.0 PL=0
MOVL C00705 V=800.0 PL=0
MOVL C00706 V=800.0 PL=0
MOVL C00707 V=800.0 PL=0
MOVL C00708 V=800.0 PL=0
MOVL C00709 V=800.0 PL=0
MOVL C00710 V=800.0 PL=0
MOVL C00711 V=800.0 PL=0
MOVL C00712 V=800.0 PL=0
MOVL C00713 V=800.0 PL=0
MOVL C00714 V=800.0 PL=0
MOVL C00715 V=800.0 PL=0
MOVL C00716 V=800.0 PL=0
MOVL C00717 V=800.0 PL=0
MOVL C00718 V=800.0 PL=0
MOVL C00719 V=800.0 PL=0
MOVL C00720 V=800.0 PL=0
MOVL C00721 V=800.0 PL=0
MOVL C00722 V=800.0 PL=0
MOVL C00723 V=800.0 PL=0
MOVL C00724 V=800.0 PL=0
MOVL C00725 V=800.0 PL=0
MOVL C00726 V=800.0 PL=0
MOVL C00727 V=800.0 PL=0
MOVL C00728 V=800.0 PL=0
MOVL C00729 V=800.0 PL=0
MOVL C00730 V=800.0 PL=0
MOVL C00731 V=800.0 PL=0
MOVL C00732 V=800.0 PL=0
MOVL C00733 V=800.0 PL=0
MOVL C00734 V=800.0 PL=0
MOVL C00735 V=800.0 PL=0
MOVL C00736 V=800.0 PL=0
MOVL C00737 V=800.0 PL=0
MOVL C00738 V=800.0 PL=0
MOVL C00739 V=800.0 PL=0
MOVL C00740 V=800.0 PL=0
MOVL C00741 V=800.0 PL=0
MOVL C00742 V=800.0 PL=0
MOVL C00743 V=800.0 PL=0
MOVL C00744 V=800.0 PL=0
MOVL C00745 V=800.0 PL=0
MOVL C00746 V=800.0 PL=0
MOVL C00747 V=800.0 PL=0
MOVL C00748 V=800.0 PL=0
MOVL C00749 V=800.0 PL=0
MOVL C00750 V=800.0 PL=0
MOVL C00751 V=800.0 PL=0
MOVL C00752 V=800.0 PL=0
MOVL C00753 V=800.0 PL=0
MOVL C00754 V=800.0 PL=0
MOVL C00755 V=800.0 PL=0
MOVL C00756 V=800.0 PL=0
MOVL C00757 V=800.0 PL=0
MOVL C00758 V=800.0 PL=0
MOVL C00759 V=800.0 PL=0
MOVL C00760 V=800.0 PL=0
MOVL C00761 V=800.0 PL=0
MOVL C00762 V=800.0 PL=0
MOVL C00763 V=800.0 PL=0
MOVL C00764 V=800.0 PL=0
MOVL C00765 V=800.0 PL=0
MOVL C00766 V=800.0 PL=0
MOVL C00767 V=800.0 PL=0
MOVL C00768 V=800.0 PL=0
MOVL C00769 V=800.0 PL=0
MOVL C00770 V=800.0 PL=0
MOVL C00771 V=800.0 PL=0
MOVL C00772 V=800.0 PL=0
MOVL C00773 V=800.0 PL=0
MOVL C00774 V=800.0 PL=0
MOVL C00775 V=800.0 PL=0
MOVL C00776 V=800.0 PL=0
MOVL C00777 V=800.0 PL=0
MOVL C00778 V=800.0 PL=0
MOVL C00779 V=800.0 PL=0
MOVL C00780 V=800.0 PL=0
MOVL C00781 V=800.0 PL=0
MOVL C00782 V=800.0 PL=0
MOVL C00783 V=800.0 PL=0
MOVL C00784 V=800.0 PL=0
MOVL C00785 V=800.0 PL=0
MOVL C00786 V=800.0 PL=0
MOVL C00787 V=800.0 PL=0
MOVL C00788 V=800.0 PL=0
MOVL C00789 V=800.0 PL=0
MOVL C00790 V=800.0 PL=0
MOVL C00791 V=800.0 PL=0
MOVL C00792 V=800.0 PL=0
MOVL C00793 V=800.0 PL=0
MOVL C00794 V=800.0 PL=0
MOVL C00795 V=800.0 PL=0
MOVL C00796 V=800.0 PL=0
MOVL C00797 V=800.0 PL=0
MOVL C00798 V=800.0 PL=0
MOVL C00799 V=800.0 PL=0
MOVL C00800 V=800.0 PL=0
MOVL C00801 V=800.0 PL=0
MOVL C00802 V=800.0 PL=0
MOVL C00803 V=800.0 PL=0
MOVL C00804 V=800.0 PL=0
MOVL C00805 V=800.0 PL=0
MOVL C00806 V=800.0 PL=0
MOVL C00807 V=800.0 PL=0
MOVL C00808 V=800.0 PL=0
MOVL C00809 V=800.0 PL=0
MOVL C00810 V=800.0 PL=0
MOVL C00811 V=800.0 PL=0
MOVL C00812 V=800.0 PL=0
MOVL C00813 V=800.0 PL=0
MOVL C00814 V=800.0 PL=0
MOVL C00815 V=800.0 PL=0
MOVL C00816 V=800.0 PL=0
MOVL C00817 V=800.0 PL=0
MOVL C00818 V=800.0 PL=0
MOVL C00819 V=800.0 PL=0
MOVL C00820 V=800.0 PL=0
MOVL C00821 V=800.0 PL=0
MOVL C00822 V=800.0 PL=0
MOVL C00823 V=800.0 PL=0
MOVL C00824 V=800.0 PL=0
MOVL C00825 V=800.0 PL=0
MOVL C00826 V=800.0 PL=0
MOVL C00827 V=800.0 PL=0
MOVL C00828 V=800.0 PL=0
MOVL C00829 V=800.0 PL=0
MOVL C00830 V=800.0 PL=0
MOVL C00831 V=800.0 PL=0
MOVL C00832 V=800.0 PL=0
MOVL C00833 V=800.0 PL=0
MOVL C00834 V=800.0 PL=0
MOVL C00835 V=800.0 PL=0
MOVL C00836 V=800.0 PL=0
MOVL C00837 V=800.0 PL=0
MOVL C00838 V=800.0 PL=0
MOVL C00839 V=800.0 PL=0
MOVL C00840 V=800.0 PL=0
MOVL C00841 V=800.0 PL=0
MOVL C00842 V=800.0 PL=0
MOVL C00843 V=800.0 PL=0
MOVL C00844 V=800.0 PL=0
MOVL C00845 V=800.0 PL=0
MOVL C00846 V=800.0 PL=0
MOVL C00847 V=800.0 PL=0
MOVL C00848 V=800.0 PL=0
MOVL C00849 V=800.0 PL=0
MOVL C00850 V=800.0 PL=0
MOVL C00851 V=800.0 PL=0
MOVL C00852 V=800.0 PL=0
MOVL C00853 V=800.0 PL=0
MOVL C00854 V=800.0 PL=0
MOVL C00855 V=800.0 PL=0
MOVL C00856 V=800.0 PL=0
MOVL C00857 V=800.0 PL=0
MOVL C00858 V=800.0 PL=0
MOVL C00859 V=800.0 PL=0
MOVL C00860 V=800.0 PL=0
MOVL C00861 V=800.0 PL=0
MOVL C00862 V=800.0 PL=0
MOVL C00863 V=800.0 PL=0
MOVL C00864 V=800.0 PL=0
MOVL C00865 V=800.0 PL=0
MOVL C00866 V=800.0 PL=0
MOVL C00867 V=800.0 PL=0
MOVL C00868 V=800.0 PL=0
MOVL C00869 V=800.0 PL=0
MOVL C00870 V=800.0 PL=0
MOVL C00871 V=800.0 PL=0
MOVL C00872 V=800.0 PL=0
MOVL C00873 V=800.0 PL=0
MOVL C00874 V=800.0 PL=0
MOVL C00875 V=800.0 PL=0
MOVL C00876 V=800.0 PL=0
MOVL C00877 V=800.0 PL=0
MOVL C00878 V=800.0 PL=0
MOVL C00879 V=800.0 PL=0
MOVL C00880 V=800.0 PL=0
MOVL C00881 V=800.0 PL=0
MOVL C00882 V=800.0 PL=0
MOVL C00883 V=800.0 PL=0
MOVL C00884 V=800.0 PL=0
MOVL C00885 V=800.0 PL=0
MOVL C00886 V=800.0 PL=0
MOVL C00887 V=800.0 PL=0
MOVL C00888 V=800.0 PL=0
MOVL C00889 V=800.0 PL=0
MOVL C00890 V=800.0 PL=0
MOVL C00891 V=800.0 PL=0
MOVL C00892 V=800.0 PL=0
MOVL C00893 V=800.0 PL=0
MOVL C00894 V=800.0 PL=0
MOVL C00895 V=800.0 PL=0
MOVL C00896 V=800.0 PL=0
MOVL C00897 V=800.0 PL=0
MOVL C00898 V=800.0 PL=0
MOVL C00899 V=800.0 PL=0
MOVL C00900 V=800.0 PL=0
MOVL C00901 V=800.0 PL=0
MOVL C00902 V=800.0 PL=0
MOVL C00903 V=800.0 PL=0
MOVL C00904 V=800.0 PL=0
MOVL C00905 V=800.0 PL=0
MOVL C00906 V=800.0 PL=0
MOVL C00907 V=800.0 PL=0
MOVL C00908 V=800.0 PL=0
MOVL C00909 V=800.0 PL=0
MOVL C00910 V=800.0 PL=0
MOVL C00911 V=800.0 PL=0
MOVL C00912 V=800.0 PL=0
MOVL C00913 V=800.0 PL=0
MOVL C00914 V=800.0 PL=0
MOVL C00915 V=800.0 PL=0
MOVL C00916 V=800.0 PL=0
MOVL C00917 V=800.0 PL=0
MOVL C00918 V=800.0 PL=0
MOVL C00919 V=800.0 PL=0
MOVL C00920 V=800.0 PL=0
MOVL C00921 V=800.0 PL=0
MOVL C00922 V=800.0 PL=0
MOVL C00923 V=800.0 PL=0
MOVL C00924 V=800.0 PL=0
MOVL C00925 V=800.0 PL=0
MOVL C00926 V=800.0 PL=0
MOVL C00927 V=800.0 PL=0
MOVL C00928 V=800.0 PL=0
MOVL C00929 V=800.0 PL=0
MOVL C00930 V=800.0 PL=0
MOVL C00931 V=800.0 PL=0
MOVL C00932 V=800.0 PL=0
MOVL C00933 V=800.0 PL=0
MOVL C00934 V=800.0 PL=0
MOVL C00935 V=800.0 PL=0
MOVL C00936 V=800.0 PL=0
MOVL C00937 V=800.0 PL=0
MOVL C00938 V=800.0 PL=0
MOVL C00939 V=800.0 PL=0
MOVL C00940 V=800.0 PL=0
MOVL C00941 V=800.0 PL=0
MOVL C00942 V=800.0 PL=0
MOVL C00943 V=800.0 PL=0
MOVL C00944 V=800.0 PL=0
MOVL C00945 V=800.0 PL=0
MOVL C00946 V=800.0 PL=0
MOVL C00947 V=800.0 PL=0
MOVL C00948 V=800.0 PL=0
MOVL C00949 V=800.0 PL=0
MOVL C00950 V=800.0 PL=0
MOVL C00951 V=800.0 PL=0
MOVL C00952 V=800.0 PL=0
MOVL C00953 V=800.0 PL=0
MOVL C00954 V=800.0 PL=0
MOVL C00955 V=800.0 PL=0
MOVL C00956 V=800.0 PL=0
MOVL C00957 V=800.0 PL=0
MOVL C00958 V=800.0 PL=0
MOVL C00959 V=800.0 PL=0
MOVL C00960 V=800.0 PL=0
MOVL C00961 V=800.0 PL=0
MOVL C00962 V=800.0 PL=0
MOVL C00963 V=800.0 PL=0
MOVL C00964 V=800.0 PL=0
MOVL C00965 V=800.0 PL=0
MOVL C00966 V=800.0 PL=0
MOVL C00967 V=800.0 PL=0
MOVL C00968 V=800.0 PL=0
MOVL C00969 V=800.0 PL=0
MOVL C00970 V=800.0 PL=0
MOVL C00971 V=800.0 PL=0
MOVL C00972 V=800.0 PL=0
MOVL C00973 V=800.0 PL=0
MOVL C00974 V=800.0 PL=0
MOVL C00975 V=800.0 PL=0
MOVL C00976 V=800.0 PL=0
MOVL C00977 V=800.0 PL=0
MOVL C00978 V=800.0 PL=0
MOVL C00979 V=800.0 PL=0
MOVL C00980 V=800.0 PL=0
MOVL C00981 V=800.0 PL=0
MOVL C00982 V=800.0 PL=0
MOVL C00983 V=800.0 PL=0
MOVL C00984 V=800.0 PL=0
MOVL C00985 V=800.0 PL=0
MOVL C00986 V=800.0 PL=0
MOVL C00987 V=800.0 PL=0
MOVL C00988 V=800.0 PL=0
MOVL C00989 V=800.0 PL=0
MOVL C00990 V=800.0 PL=0
MOVL C00991 V=800.0 PL=0
MOVL C00992 V=800.0 PL=0
MOVL C00993 V=800.0 PL=0
MOVL C00994 V=800.0 PL=0
MOVL C00995 V=800.0 PL=0
MOVL C00996 V=800.0 PL=0
MOVL C00997 V=800.0 PL=0
MOVL C00998 V=800.0 PL=0
MOVL C00999 V=800.0 PL=0
MOVL C01000 V=800.0 PL=0
MOVL C01001 V=800.0 PL=0
MOVL C01002 V=800.0 PL=0
MOVL C01003 V=800.0 PL=0
MOVL C01004 V=800.0 PL=0
MOVL C01005 V=800.0 PL=0
MOVL C01006 V=800.0 PL=0
MOVL C01007 V=800.0 PL=0
MOVL C01008 V=800.0 PL=0
MOVL C01009 V=800.0 PL=0
MOVL C01010 V=800.0 PL=0
MOVL C01011 V=800.0 PL=0
MOVL C01012 V=800.0 PL=0
MOVL C01013 V=800.0 PL=0
MOVL C01014 V=800.0 PL=0
MOVL C01015 V=800.0 PL=0
MOVL C01016 V=800.0 PL=0
MOVL C01017 V=800.0 PL=0
MOVL C01018 V=800.0 PL=0
MOVL C01019 V=800.0 PL=0
MOVL C01020 V=800.0 PL=0
MOVL C01021 V=800.0 PL=0
MOVL C01022 V=800.0 PL=0
MOVL C01023 V=800.0 PL=0
MOVL C01024 V=800.0 PL=0
MOVL C01025 V=800.0 PL=0
MOVL C01026 V=800.0 PL=0
MOVL C01027 V=800.0 PL=0
MOVL C01028 V=800.0 PL=0
MOVL C01029 V=800.0 PL=0
MOVL C01030 V=800.0 PL=0
MOVL C01031 V=800.0 PL=0
MOVL C01032 V=800.0 PL=0
MOVL C01033 V=800.0 PL=0
MOVL C01034 V=800.0 PL=0
MOVL C01035 V=800.0 PL=0
MOVL C01036 V=800.0 PL=0
MOVL C01037 V=800.0 PL=0
MOVL C01038 V=800.0 PL=0
MOVL C01039 V=800.0 PL=0
MOVL C01040 V=800.0 PL=0
MOVL C01041 V=800.0 PL=0
MOVL C01042 V=800.0 PL=0
MOVL C01043 V=800.0 PL=0
MOVL C01044 V=800.0 PL=0
MOVL C01045 V=800.0 PL=0
MOVL C01046 V=800.0 PL=0
MOVL C01047 V=800.0 PL=0
MOVL C01048 V=800.0 PL=0
MOVL C01049 V=800.0 PL=0
MOVL C01050 V=800.0 PL=0
MOVL C01051 V=800.0 PL=0
MOVL C01052 V=800.0 PL=0
MOVL C01053 V=800.0 PL=0
MOVL C01054 V=800.0 PL=0
MOVL C01055 V=800.0 PL=0
MOVL C01056 V=800.0 PL=0
MOVL C01057 V=800.0 PL=0
MOVL C01058 V=800.0 PL=0
MOVL C01059 V=800.0 PL=0
MOVL C01060 V=800.0 PL=0
MOVL C01061 V=800.0 PL=0
MOVL C01062 V=800.0 PL=0
MOVL C01063 V=800.0 PL=0
MOVL C01064 V=800.0 PL=0
MOVL C01065 V=800.0 PL=0
MOVL C01066 V=800.0 PL=0
MOVL C01067 V=800.0 PL=0
MOVL C01068 V=800.0 PL=0
MOVL C01069 V=800.0 PL=0
MOVL C01070 V=800.0 PL=0
MOVL C01071 V=800.0 PL=0
MOVL C01072 V=800.0 PL=0
MOVL C01073 V=800.0 PL=0
MOVL C01074 V=800.0 PL=0
MOVL C01075 V=800.0 PL=0
MOVL C01076 V=800.0 PL=0
MOVL C01077 V=800.0 PL=0
MOVL C01078 V=800.0 PL=0
MOVL C01079 V=800.0 PL=0
MOVL C01080 V=800.0 PL=0
MOVL C01081 V=800.0 PL=0
MOVL C01082 V=800.0 PL=0
MOVL C01083 V=800.0 PL=0
MOVL C01084 V=800.0 PL=0
MOVL C01085 V=800.0 PL=0
MOVL C01086 V=800.0 PL=0
MOVL C01087 V=800.0 PL=0
MOVL C01088 V=800.0 PL=0
MOVL C01089 V=800.0 PL=0
MOVL C01090 V=800.0 PL=0
MOVL C01091 V=800.0 PL=0
MOVL C01092 V=800.0 PL=0
MOVL C01093 V=800.0 PL=0
MOVL C01094 V=800.0 PL=0
MOVL C01095 V=800.0 PL=0
MOVL C01096 V=800.0 PL=0
MOVL C01097 V=800.0 PL=0
MOVL C01098 V=800.0 PL=0
MOVL C01099 V=800.0 PL=0
MOVL C01100 V=800.0 PL=0
MOVL C01101 V=800.0 PL=0
MOVL C01102 V=800.0 PL=0
MOVL C01103 V=800.0 PL=0
MOVL C01104 V=800.0 PL=0
MOVL C01105 V=800.0 PL=0
MOVL C01106 V=800.0 PL=0
MOVL C01107 V=800.0 PL=0
MOVL C01108 V=800.0 PL=0
MOVL C01109 V=800.0 PL=0
MOVL C01110 V=800.0 PL=0
MOVL C01111 V=800.0 PL=0
MOVL C01112 V=800.0 PL=0
MOVL C01113 V=800.0 PL=0
MOVL C01114 V=800.0 PL=0
MOVL C01115 V=800.0 PL=0
MOVL C01116 V=800.0 PL=0
MOVL C01117 V=800.0 PL=0
MOVL C01118 V=800.0 PL=0
MOVL C01119 V=800.0 PL=0
MOVL C01120 V=800.0 PL=0
MOVL C01121 V=800.0 PL=0
MOVL C01122 V=800.0 PL=0
MOVL C01123 V=800.0 PL=0
MOVL C01124 V=800.0 PL=0
MOVL C01125 V=800.0 PL=0
MOVL C01126 V=800.0 PL=0
MOVL C01127 V=800.0 PL=0
MOVL C01128 V=800.0 PL=0
MOVL C01129 V=800.0 PL=0
MOVL C01130 V=800.0 PL=0
MOVL C01131 V=800.0 PL=0
MOVL C01132 V=800.0 PL=0
MOVL C01133 V=800.0 PL=0
MOVL C01134 V=800.0 PL=0
MOVL C01135 V=800.0 PL=0
MOVL C01136 V=800.0 PL=0
MOVL C01137 V=800.0 PL=0
MOVL C01138 V=800.0 PL=0
MOVL C01139 V=800.0 PL=0
MOVL C01140 V=800.0 PL=0
MOVL C01141 V=800.0 PL=0
MOVL C01142 V=800.0 PL=0
MOVL C01143 V=800.0 PL=0
MOVL C01144 V=800.0 PL=0
MOVL C01145 V=800.0 PL=0
MOVL C01146 V=800.0 PL=0
MOVL C01147 V=800.0 PL=0
MOVL C01148 V=800.0 PL=0
MOVL C01149 V=800.0 PL=0
MOVL C01150 V=800.0 PL=0
MOVL C01151 V=800.0 PL=0
MOVL C01152 V=800.0 PL=0
MOVL C01153 V=800.0 PL=0
MOVL C01154 V=800.0 PL=0
MOVL C01155 V=800.0 PL=0
MOVL C01156 V=800.0 PL=0
MOVL C01157 V=800.0 PL=0
MOVL C01158 V=800.0 PL=0
MOVL C01159 V=800.0 PL=0
MOVL C01160 V=800.0 PL=0
MOVL C01161 V=800.0 PL=0
MOVL C01162 V=800.0 PL=0
MOVL C01163 V=800.0 PL=0
MOVL C01164 V=800.0 PL=0
MOVL C01165 V=800.0 PL=0
MOVL C01166 V=800.0 PL=0
MOVL C01167 V=800.0 PL=0
MOVL C01168 V=800.0 PL=0
MOVL C01169 V=800.0 PL=0
MOVL C01170 V=800.0 PL=0
MOVL C01171 V=800.0 PL=0
MOVL C01172 V=800.0 PL=0
MOVL C01173 V=800.0 PL=0
MOVL C01174 V=800.0 PL=0
MOVL C01175 V=800.0 PL=0
MOVL C01176 V=800.0 PL=0
MOVL C01177 V=800.0 PL=0
MOVL C01178 V=800.0 PL=0
MOVL C01179 V=800.0 PL=0
MOVL C01180 V=800.0 PL=0
MOVL C01181 V=800.0 PL=0
MOVL C01182 V=800.0 PL=0
MOVL C01183 V=800.0 PL=0
MOVL C01184 V=800.0 PL=0
MOVL C01185 V=800.0 PL=0
MOVL C01186 V=800.0 PL=0
MOVL C01187 V=800.0 PL=0
MOVL C01188 V=800.0 PL=0
MOVL C01189 V=800.0 PL=0
MOVL C01190 V=800.0 PL=0
MOVL C01191 V=800.0 PL=0
MOVL C01192 V=800.0 PL=0
MOVL C01193 V=800.0 PL=0
MOVL C01194 V=800.0 PL=0
MOVL C01195 V=800.0 PL=0
MOVL C01196 V=800.0 PL=0
MOVL C01197 V=800.0 PL=0
MOVL C01198 V=800.0 PL=0
MOVL C01199 V=800.0 PL=0
MOVL C01200 V=800.0 PL=0
MOVL C01201 V=800.0 PL=0
MOVL C01202 V=800.0 PL=0
MOVL C01203 V=800.0 PL=0
MOVL C01204 V=800.0 PL=0
MOVL C01205 V=800.0 PL=0
MOVL C01206 V=800.0 PL=0
MOVL C01207 V=800.0 PL=0
MOVL C01208 V=800.0 PL=0
MOVL C01209 V=800.0 PL=0
MOVL C01210 V=800.0 PL=0
MOVL C01211 V=800.0 PL=0
MOVL C01212 V=800.0 PL=0
MOVL C01213 V=800.0 PL=0
MOVL C01214 V=800.0 PL=0
MOVL C01215 V=800.0 PL=0
MOVL C01216 V=800.0 PL=0
MOVL C01217 V=800.0 PL=0
MOVL C01218 V=800.0 PL=0
MOVL C01219 V=800.0 PL=0
MOVL C01220 V=800.0 PL=0
MOVL C01221 V=800.0 PL=0
MOVL C01222 V=800.0 PL=0
MOVL C01223 V=800.0 PL=0
MOVL C01224 V=800.0 PL=0
MOVL C01225 V=800.0 PL=0
MOVL C01226 V=800.0 PL=0
MOVL C01227 V=800.0 PL=0
MOVL C01228 V=800.0 PL=0
MOVL C01229 V=800.0 PL=0
MOVL C01230 V=800.0 PL=0
MOVL C01231 V=800.0 PL=0
MOVL C01232 V=800.0 PL=0
MOVL C01233 V=800.0 PL=0
MOVL C01234 V=800.0 PL=0
MOVL C01235 V=800.0 PL=0
MOVL C01236 V=800.0 PL=0
MOVL C01237 V=800.0 PL=0
MOVL C01238 V=800.0 PL=0
MOVL C01239 V=800.0 PL=0
MOVL C01240 V=800.0 PL=0
MOVL C01241 V=800.0 PL=0
MOVL C01242 V=800.0 PL=0
MOVL C01243 V=800.0 PL=0
MOVL C01244 V=800.0 PL=0
MOVL C01245 V=800.0 PL=0
MOVL C01246 V=800.0 PL=0
MOVL C01247 V=800.0 PL=0
MOVL C01248 V=800.0 PL=0
MOVL C01249 V=800.0 PL=0
MOVL C01250 V=800.0 PL=0
MOVL C01251 V=800.0 PL=0
MOVL C01252 V=800.0 PL=0
MOVL C01253 V=800.0 PL=0
MOVL C01254 V=800.0 PL=0
MOVL C01255 V=800.0 PL=0
MOVL C01256 V=800.0 PL=0
MOVL C01257 V=800.0 PL=0
MOVL C01258 V=800.0 PL=0
MOVL C01259 V=800.0 PL=0
MOVL C01260 V=800.0 PL=0
MOVL C01261 V=800.0 PL=0
MOVL C01262 V=800.0 PL=0
MOVL C01263 V=800.0 PL=0
MOVL C01264 V=800.0 PL=0
MOVL C01265 V=800.0 PL=0
MOVL C01266 V=800.0 PL=0
MOVL C01267 V=800.0 PL=0
MOVL C01268 V=800.0 PL=0
MOVL C01269 V=800.0 PL=0
MOVL C01270 V=800.0 PL=0
MOVL C01271 V=800.0 PL=0
MOVL C01272 V=800.0 PL=0
MOVL C01273 V=800.0 PL=0
MOVL C01274 V=800.0 PL=0
MOVL C01275 V=800.0 PL=0
MOVL C01276 V=800.0 PL=0
MOVL C01277 V=800.0 PL=0
MOVL C01278 V=800.0 PL=0
MOVL C01279 V=800.0 PL=0
MOVL C01280 V=800.0 PL=0
MOVL C01281 V=800.0 PL=0
MOVL C01282 V=800.0 PL=0
MOVL C01283 V=800.0 PL=0
MOVL C01284 V=800.0 PL=0
MOVL C01285 V=800.0 PL=0
MOVL C01286 V=800.0 PL=0
MOVL C01287 V=800.0 PL=0
MOVL C01288 V=800.0 PL=0
MOVL C01289 V=800.0 PL=0
MOVL C01290 V=800.0 PL=0
MOVL C01291 V=800.0 PL=0
MOVL C01292 V=800.0 PL=0
MOVL C01293 V=800.0 PL=0
MOVL C01294 V=800.0 PL=0
MOVL C01295 V=800.0 PL=0
MOVL C01296 V=800.0 PL=0
MOVL C01297 V=800.0 PL=0
MOVL C01298 V=800.0 PL=0
MOVL C01299 V=800.0 PL=0
MOVL C01300 V=800.0 PL=0
MOVL C01301 V=800.0 PL=0
MOVL C01302 V=800.0 PL=0
MOVL C01303 V=800.0 PL=0
MOVL C01304 V=800.0 PL=0
MOVL C01305 V=800.0 PL=0
MOVL C01306 V=800.0 PL=0
MOVL C01307 V=800.0 PL=0
MOVL C01308 V=800.0 PL=0
MOVL C01309 V=800.0 PL=0
MOVL C01310 V=800.0 PL=0
MOVL C01311 V=800.0 PL=0
MOVL C01312 V=800.0 PL=0
MOVL C01313 V=800.0 PL=0
MOVL C01314 V=800.0 PL=0
MOVL C01315 V=800.0 PL=0
MOVL C01316 V=800.0 PL=0
MOVL C01317 V=800.0 PL=0
MOVL C01318 V=800.0 PL=0
MOVL C01319 V=800.0 PL=0
MOVL C01320 V=800.0 PL=0
MOVL C01321 V=800.0 PL=0
MOVL C01322 V=800.0 PL=0
MOVL C01323 V=800.0 PL=0
MOVL C01324 V=800.0 PL=0
MOVL C01325 V=800.0 PL=0
MOVL C01326 V=800.0 PL=0
MOVL C01327 V=800.0 PL=0
MOVL C01328 V=800.0 PL=0
MOVL C01329 V=800.0 PL=0
MOVL C01330 V=800.0 PL=0
MOVL C01331 V=800.0 PL=0
MOVL C01332 V=800.0 PL=0
MOVL C01333 V=800.0 PL=0
MOVL C01334 V=800.0 PL=0
MOVL C01335 V=800.0 PL=0
MOVL C01336 V=800.0 PL=0
MOVL C01337 V=800.0 PL=0
MOVL C01338 V=800.0 PL=0
MOVL C01339 V=800.0 PL=0
MOVL C01340 V=800.0 PL=0
MOVL C01341 V=800.0 PL=0
MOVL C01342 V=800.0 PL=0
MOVL C01343 V=800.0 PL=0
MOVL C01344 V=800.0 PL=0
MOVL C01345 V=800.0 PL=0
MOVL C01346 V=800.0 PL=0
MOVL C01347 V=800.0 PL=0
MOVL C01348 V=800.0 PL=0
MOVL C01349 V=800.0 PL=0
MOVL C01350 V=800.0 PL=0
MOVL C01351 V=800.0 PL=0
MOVL C01352 V=800.0 PL=0
MOVL C01353 V=800.0 PL=0
MOVL C01354 V=800.0 PL=0
MOVL C01355 V=800.0 PL=0
MOVL C01356 V=800.0 PL=0
MOVL C01357 V=800.0 PL=0
MOVL C01358 V=800.0 PL=0
MOVL C01359 V=800.0 PL=0
MOVL C01360 V=800.0 PL=0
MOVL C01361 V=800.0 PL=0
MOVL C01362 V=800.0 PL=0
MOVL C01363 V=800.0 PL=0
MOVL C01364 V=800.0 PL=0
MOVL C01365 V=800.0 PL=0
MOVL C01366 V=800.0 PL=0
MOVL C01367 V=800.0 PL=0
MOVL C01368 V=800.0 PL=0
MOVL C01369 V=800.0 PL=0
MOVL C01370 V=800.0 PL=0
MOVL C01371 V=800.0 PL=0
MOVL C01372 V=800.0 PL=0
MOVL C01373 V=800.0 PL=0
MOVL C01374 V=800.0 PL=0
MOVL C01375 V=800.0 PL=0
MOVL C01376 V=800.0 PL=0
MOVL C01377 V=800.0 PL=0
MOVL C01378 V=800.0 PL=0
MOVL C01379 V=800.0 PL=0
MOVL C01380 V=800.0 PL=0
MOVL C01381 V=800.0 PL=0
MOVL C01382 V=800.0 PL=0
MOVL C01383 V=800.0 PL=0
MOVL C01384 V=800.0 PL=0
MOVL C01385 V=800.0 PL=0
MOVL C01386 V=800.0 PL=0
MOVL C01387 V=800.0 PL=0
MOVL C01388 V=800.0 PL=0
MOVL C01389 V=800.0 PL=0
MOVL C01390 V=800.0 PL=0
MOVL C01391 V=800.0 PL=0
MOVL C01392 V=800.0 PL=0
MOVL C01393 V=800.0 PL=0
MOVL C01394 V=800.0 PL=0
MOVL C01395 V=800.0 PL=0
MOVL C01396 V=800.0 PL=0
MOVL C01397 V=800.0 PL=0
MOVL C01398 V=800.0 PL=0
MOVL C01399 V=800.0 PL=0
MOVL C01400 V=800.0 PL=0
MOVL C01401 V=800.0 PL=0
MOVL C01402 V=800.0 PL=0
MOVL C01403 V=800.0 PL=0
MOVL C01404 V=800.0 PL=0
MOVL C01405 V=800.0 PL=0
MOVL C01406 V=800.0 PL=0
MOVL C01407 V=800.0 PL=0
MOVL C01408 V=800.0 PL=0
MOVL C01409 V=800.0 PL=0
MOVL C01410 V=800.0 PL=0
MOVL C01411 V=800.0 PL=0
MOVL C01412 V=800.0 PL=0
MOVL C01413 V=800.0 PL=0
MOVL C01414 V=800.0 PL=0
MOVL C01415 V=800.0 PL=0
MOVL C01416 V=800.0 PL=0
MOVL C01417 V=800.0 PL=0
MOVL C01418 V=800.0 PL=0
MOVL C01419 V=800.0 PL=0
MOVL C01420 V=800.0 PL=0
MOVL C01421 V=800.0 PL=0
MOVL C01422 V=800.0 PL=0
MOVL C01423 V=800.0 PL=0
MOVL C01424 V=800.0 PL=0
MOVL C01425 V=800.0 PL=0
MOVL C01426 V=800.0 PL=0
MOVL C01427 V=800.0 PL=0
MOVL C01428 V=800.0 PL=0
MOVL C01429 V=800.0 PL=0
MOVL C01430 V=800.0 PL=0
MOVL C01431 V=800.0 PL=0
MOVL C01432 V=800.0 PL=0
MOVL C01433 V=800.0 PL=0
MOVL C01434 V=800.0 PL=0
MOVL C01435 V=800.0 PL=0
MOVL C01436 V=800.0 PL=0
MOVL C01437 V=800.0 PL=0
MOVL C01438 V=800.0 PL=0
MOVL C01439 V=800.0 PL=0
MOVL C01440 V=800.0 PL=0
MOVL C01441 V=800.0 PL=0
MOVL C01442 V=800.0 PL=0
MOVL C01443 V=800.0 PL=0
MOVL C01444 V=800.0 PL=0
MOVL C01445 V=800.0 PL=0
MOVL C01446 V=800.0 PL=0
MOVL C01447 V=800.0 PL=0
MOVL C01448 V=800.0 PL=0
MOVL C01449 V=800.0 PL=0
MOVL C01450 V=800.0 PL=0
MOVL C01451 V=800.0 PL=0
MOVL C01452 V=800.0 PL=0
MOVL C01453 V=800.0 PL=0
MOVL C01454 V=800.0 PL=0
MOVL C01455 V=800.0 PL=0
MOVL C01456 V=800.0 PL=0
MOVL C01457 V=800.0 PL=0
MOVL C01458 V=800.0 PL=0
MOVL C01459 V=800.0 PL=0
MOVL C01460 V=800.0 PL=0
MOVL C01461 V=800.0 PL=0
MOVL C01462 V=800.0 PL=0
MOVL C01463 V=800.0 PL=0
MOVL C01464 V=800.0 PL=0
MOVL C01465 V=800.0 PL=0
MOVL C01466 V=800.0 PL=0
MOVL C01467 V=800.0 PL=0
MOVL C01468 V=800.0 PL=0
MOVL C01469 V=800.0 PL=0
MOVL C01470 V=800.0 PL=0
MOVL C01471 V=800.0 PL=0
MOVL C01472 V=800.0 PL=0
MOVL C01473 V=800.0 PL=0
MOVL C01474 V=800.0 PL=0
MOVL C01475 V=800.0 PL=0
MOVL C01476 V=800.0 PL=0
MOVL C01477 V=800.0 PL=0
MOVL C01478 V=800.0 PL=0
MOVL C01479 V=800.0 PL=0
MOVL C01480 V=800.0 PL=0
MOVL C01481 V=800.0 PL=0
MOVL C01482 V=800.0 PL=0
MOVL C01483 V=800.0 PL=0
MOVL C01484 V=800.0 PL=0
MOVL C01485 V=800.0 PL=0
MOVL C01486 V=800.0 PL=0
MOVL C01487 V=800.0 PL=0
MOVL C01488 V=800.0 PL=0
MOVL C01489 V=800.0 PL=0
MOVL C01490 V=800.0 PL=0
MOVL C01491 V=800.0 PL=0
MOVL C01492 V=800.0 PL=0
MOVL C01493 V=800.0 PL=0
MOVL C01494 V=800.0 PL=0
MOVL C01495 V=800.0 PL=0
MOVL C01496 V=800.0 PL=0
MOVL C01497 V=800.0 PL=0
MOVL C01498 V=800.0 PL=0
MOVL C01499 V=800.0 PL=0
MOVL C01500 V=800.0 PL=0
MOVL C01501 V=800.0 PL=0
MOVL C01502 V=800.0 PL=0
MOVL C01503 V=800.0 PL=0
MOVL C01504 V=800.0 PL=0
MOVL C01505 V=800.0 PL=0
MOVL C01506 V=800.0 PL=0
MOVL C01507 V=800.0 PL=0
MOVL C01508 V=800.0 PL=0
MOVL C01509 V=800.0 PL=0
MOVL C01510 V=800.0 PL=0
MOVL C01511 V=800.0 PL=0
MOVL C01512 V=800.0 PL=0
MOVL C01513 V=800.0 PL=0
MOVL C01514 V=800.0 PL=0
MOVL C01515 V=800.0 PL=0
MOVL C01516 V=800.0 PL=0
MOVL C01517 V=800.0 PL=0
MOVL C01518 V=800.0 PL=0
MOVL C01519 V=800.0 PL=0
MOVL C01520 V=800.0 PL=0
MOVL C01521 V=800.0 PL=0
MOVL C01522 V=800.0 PL=0
MOVL C01523 V=800.0 PL=0
MOVL C01524 V=800.0 PL=0
MOVL C01525 V=800.0 PL=0
MOVL C01526 V=800.0 PL=0
MOVL C01527 V=800.0 PL=0
MOVL C01528 V=800.0 PL=0
MOVL C01529 V=800.0 PL=0
MOVL C01530 V=800.0 PL=0
MOVL C01531 V=800.0 PL=0
MOVL C01532 V=800.0 PL=0
MOVL C01533 V=800.0 PL=0
MOVL C01534 V=800.0 PL=0
MOVL C01535 V=800.0 PL=0
MOVL C01536 V=800.0 PL=0
MOVL C01537 V=800.0 PL=0
MOVL C01538 V=800.0 PL=0
MOVL C01539 V=800.0 PL=0
MOVL C01540 V=800.0 PL=0
MOVL C01541 V=800.0 PL=0
MOVL C01542 V=800.0 PL=0
MOVL C01543 V=800.0 PL=0
MOVL C01544 V=800.0 PL=0
MOVL C01545 V=800.0 PL=0
MOVL C01546 V=800.0 PL=0
MOVL C01547 V=800.0 PL=0
MOVL C01548 V=800.0 PL=0
MOVL C01549 V=800.0 PL=0
MOVL C01550 V=800.0 PL=0
MOVL C01551 V=800.0 PL=0
MOVL C01552 V=800.0 PL=0
MOVL C01553 V=800.0 PL=0
MOVL C01554 V=800.0 PL=0
MOVL C01555 V=800.0 PL=0
MOVL C01556 V=800.0 PL=0
MOVL C01557 V=800.0 PL=0
MOVL C01558 V=800.0 PL=0
MOVL C01559 V=800.0 PL=0
MOVL C01560 V=800.0 PL=0
MOVL C01561 V=800.0 PL=0
MOVL C01562 V=800.0 PL=0
MOVL C01563 V=800.0 PL=0
MOVL C01564 V=800.0 PL=0
MOVL C01565 V=800.0 PL=0
MOVL C01566 V=800.0 PL=0
MOVL C01567 V=800.0 PL=0
MOVL C01568 V=800.0 PL=0
MOVL C01569 V=800.0 PL=0
MOVL C01570 V=800.0 PL=0
MOVL C01571 V=800.0 PL=0
MOVL C01572 V=800.0 PL=0
MOVL C01573 V=800.0 PL=0
MOVL C01574 V=800.0 PL=0
MOVL C01575 V=800.0 PL=0
MOVL C01576 V=800.0 PL=0
MOVL C01577 V=800.0 PL=0
MOVL C01578 V=800.0 PL=0
MOVL C01579 V=800.0 PL=0
MOVL C01580 V=800.0 PL=0
MOVL C01581 V=800.0 PL=0
MOVL C01582 V=800.0 PL=0
MOVL C01583 V=800.0 PL=0
MOVL C01584 V=800.0 PL=0
MOVL C01585 V=800.0 PL=0
MOVL C01586 V=800.0 PL=0
MOVL C01587 V=800.0 PL=0
MOVL C01588 V=800.0 PL=0
MOVL C01589 V=800.0 PL=0
MOVL C01590 V=800.0 PL=0
MOVL C01591 V=800.0 PL=0
MOVL C01592 V=800.0 PL=0
MOVL C01593 V=800.0 PL=0
MOVL C01594 V=800.0 PL=0
MOVL C01595 V=800.0 PL=0
MOVL C01596 V=800.0 PL=0
MOVL C01597 V=800.0 PL=0
MOVL C01598 V=800.0 PL=0
MOVL C01599 V=800.0 PL=0
MOVL C01600 V=800.0 PL=0
MOVL C01601 V=800.0 PL=0
MOVL C01602 V=800.0 PL=0
MOVL C01603 V=800.0 PL=0
MOVL C01604 V=800.0 PL=0
MOVL C01605 V=800.0 PL=0
MOVL C01606 V=800.0 PL=0
MOVL C01607 V=800.0 PL=0
MOVL C01608 V=800.0 PL=0
MOVL C01609 V=800.0 PL=0
MOVL C01610 V=800.0 PL=0
MOVL C01611 V=800.0 PL=0
MOVL C01612 V=800.0 PL=0
MOVL C01613 V=800.0 PL=0
MOVL C01614 V=800.0 PL=0
MOVL C01615 V=800.0 PL=0
MOVL C01616 V=800.0 PL=0
MOVL C01617 V=800.0 PL=0
MOVL C01618 V=800.0 PL=0
MOVL C01619 V=800.0 PL=0
MOVL C01620 V=800.0 PL=0
MOVL C01621 V=800.0 PL=0
MOVL C01622 V=800.0 PL=0
MOVL C01623 V=800.0 PL=0
MOVL C01624 V=800.0 PL=0
MOVL C01625 V=800.0 PL=0
MOVL C01626 V=800.0 PL=0
MOVL C01627 V=800.0 PL=0
MOVL C01628 V=800.0 PL=0
MOVL C01629 V=800.0 PL=0
MOVL C01630 V=800.0 PL=0
MOVL C01631 V=800.0 PL=0
MOVL C01632 V=800.0 PL=0
MOVL C01633 V=800.0 PL=0
MOVL C01634 V=800.0 PL=0
MOVL C01635 V=800.0 PL=0
MOVL C01636 V=800.0 PL=0
MOVL C01637 V=800.0 PL=0
MOVL C01638 V=800.0 PL=0
MOVL C01639 V=800.0 PL=0
MOVL C01640 V=800.0 PL=0
MOVL C01641 V=800.0 PL=0
MOVL C01642 V=800.0 PL=0
MOVL C01643 V=800.0 PL=0
MOVL C01644 V=800.0 PL=0
MOVL C01645 V=800.0 PL=0
MOVL C01646 V=800.0 PL=0
MOVL C01647 V=800.0 PL=0
MOVL C01648 V=800.0 PL=0
MOVL C01649 V=800.0 PL=0
MOVL C01650 V=800.0 PL=0
MOVL C01651 V=800.0 PL=0
MOVL C01652 V=800.0 PL=0
MOVL C01653 V=800.0 PL=0
MOVL C01654 V=800.0 PL=0
MOVL C01655 V=800.0 PL=0
MOVL C01656 V=800.0 PL=0
MOVL C01657 V=800.0 PL=0
MOVL C01658 V=800.0 PL=0
MOVL C01659 V=800.0 PL=0
MOVL C01660 V=800.0 PL=0
MOVL C01661 V=800.0 PL=0
MOVL C01662 V=800.0 PL=0
MOVL C01663 V=800.0 PL=0
MOVL C01664 V=800.0 PL=0
MOVL C01665 V=800.0 PL=0
MOVL C01666 V=800.0 PL=0
MOVL C01667 V=800.0 PL=0
MOVL C01668 V=800.0 PL=0
MOVL C01669 V=800.0 PL=0
MOVL C01670 V=800.0 PL=0
MOVL C01671 V=800.0 PL=0
MOVL C01672 V=800.0 PL=0
MOVL C01673 V=800.0 PL=0
MOVL C01674 V=800.0 PL=0
MOVL C01675 V=800.0 PL=0
MOVL C01676 V=800.0 PL=0
MOVL C01677 V=800.0 PL=0
MOVL C01678 V=800.0 PL=0
MOVL C01679 V=800.0 PL=0
MOVL C01680 V=800.0 PL=0
MOVL C01681 V=800.0 PL=0
MOVL C01682 V=800.0 PL=0
MOVL C01683 V=800.0 PL=0
MOVL C01684 V=800.0 PL=0
MOVL C01685 V=800.0 PL=0
MOVL C01686 V=800.0 PL=0
MOVL C01687 V=800.0 PL=0
MOVL C01688 V=800.0 PL=0
MOVL C01689 V=800.0 PL=0
MOVL C01690 V=800.0 PL=0
MOVL C01691 V=800.0 PL=0
MOVL C01692 V=800.0 PL=0
MOVL C01693 V=800.0 PL=0
MOVL C01694 V=800.0 PL=0
MOVL C01695 V=800.0 PL=0
MOVL C01696 V=800.0 PL=0
MOVL C01697 V=800.0 PL=0
MOVL C01698 V=800.0 PL=0
MOVL C01699 V=800.0 PL=0
MOVL C01700 V=800.0 PL=0
MOVL C01701 V=800.0 PL=0
MOVL C01702 V=800.0 PL=0
MOVL C01703 V=800.0 PL=0
MOVL C01704 V=800.0 PL=0
MOVL C01705 V=800.0 PL=0
MOVL C01706 V=800.0 PL=0
MOVL C01707 V=800.0 PL=0
MOVL C01708 V=800.0 PL=0
MOVL C01709 V=800.0 PL=0
MOVL C01710 V=800.0 PL=0
MOVL C01711 V=800.0 PL=0
MOVL C01712 V=800.0 PL=0
MOVL C01713 V=800.0 PL=0
MOVL C01714 V=800.0 PL=0
MOVL C01715 V=800.0 PL=0
MOVL C01716 V=800.0 PL=0
MOVL C01717 V=800.0 PL=0
MOVL C01718 V=800.0 PL=0
MOVL C01719 V=800.0 PL=0
MOVL C01720 V=800.0 PL=0
MOVL C01721 V=800.0 PL=0
MOVL C01722 V=800.0 PL=0
MOVL C01723 V=800.0 PL=0
MOVL C01724 V=800.0 PL=0
MOVL C01725 V=800.0 PL=0
MOVL C01726 V=800.0 PL=0
MOVL C01727 V=800.0 PL=0
MOVL C01728 V=800.0 PL=0
MOVL C01729 V=800.0 PL=0
MOVL C01730 V=800.0 PL=0
MOVL C01731 V=800.0 PL=0
MOVL C01732 V=800.0 PL=0
MOVL C01733 V=800.0 PL=0
MOVL C01734 V=800.0 PL=0
MOVL C01735 V=800.0 PL=0
MOVL C01736 V=800.0 PL=0
MOVL C01737 V=800.0 PL=0
MOVL C01738 V=800.0 PL=0
MOVL C01739 V=800.0 PL=0
MOVL C01740 V=800.0 PL=0
MOVL C01741 V=800.0 PL=0
MOVL C01742 V=800.0 PL=0
MOVL C01743 V=800.0 PL=0
MOVL C01744 V=800.0 PL=0
MOVL C01745 V=800.0 PL=0
MOVL C01746 V=800.0 PL=0
MOVL C01747 V=800.0 PL=0
MOVL C01748 V=800.0 PL=0
MOVL C01749 V=800.0 PL=0
MOVL C01750 V=800.0 PL=0
MOVL C01751 V=800.0 PL=0
MOVL C01752 V=800.0 PL=0
MOVL C01753 V=800.0 PL=0
MOVL C01754 V=800.0 PL=0
MOVL C01755 V=800.0 PL=0
MOVL C01756 V=800.0 PL=0
MOVL C01757 V=800.0 PL=0
MOVL C01758 V=800.0 PL=0
MOVL C01759 V=800.0 PL=0
MOVL C01760 V=800.0 PL=0
MOVL C01761 V=800.0 PL=0
MOVL C01762 V=800.0 PL=0
MOVL C01763 V=800.0 PL=0
MOVL C01764 V=800.0 PL=0
MOVL C01765 V=800.0 PL=0
MOVL C01766 V=800.0 PL=0
MOVL C01767 V=800.0 PL=0
MOVL C01768 V=800.0 PL=0
MOVL C01769 V=800.0 PL=0
MOVL C01770 V=800.0 PL=0
MOVL C01771 V=800.0 PL=0
MOVL C01772 V=800.0 PL=0
MOVL C01773 V=800.0 PL=0
MOVL C01774 V=800.0 PL=0
MOVL C01775 V=800.0 PL=0
MOVL C01776 V=800.0 PL=0
MOVL C01777 V=800.0 PL=0
MOVL C01778 V=800.0 PL=0
MOVL C01779 V=800.0 PL=0
MOVL C01780 V=800.0 PL=0
MOVL C01781 V=800.0 PL=0
MOVL C01782 V=800.0 PL=0
MOVL C01783 V=800.0 PL=0
MOVL C01784 V=800.0 PL=0
MOVL C01785 V=800.0 PL=0
MOVL C01786 V=800.0 PL=0
MOVL C01787 V=800.0 PL=0
MOVL C01788 V=800.0 PL=0
MOVL C01789 V=800.0 PL=0
MOVL C01790 V=800.0 PL=0
MOVL C01791 V=800.0 PL=0
MOVL C01792 V=800.0 PL=0
MOVL C01793 V=800.0 PL=0
MOVL C01794 V=800.0 PL=0
MOVL C01795 V=800.0 PL=0
MOVL C01796 V=800.0 PL=0
MOVL C01797 V=800.0 PL=0
MOVL C01798 V=800.0 PL=0
MOVL C01799 V=800.0 PL=0
MOVL C01800 V=800.0 PL=0
MOVL C01801 V=800.0 PL=0
MOVL C01802 V=800.0 PL=0
MOVL C01803 V=800.0 PL=0
MOVL C01804 V=800.0 PL=0
MOVL C01805 V=800.0 PL=0
MOVL C01806 V=800.0 PL=0
MOVL C01807 V=800.0 PL=0
MOVL C01808 V=800.0 PL=0
MOVL C01809 V=800.0 PL=0
MOVL C01810 V=800.0 PL=0
MOVL C01811 V=800.0 PL=0
MOVL C01812 V=800.0 PL=0
MOVL C01813 V=800.0 PL=0
MOVL C01814 V=800.0 PL=0
MOVL C01815 V=800.0 PL=0
MOVL C01816 V=800.0 PL=0
MOVL C01817 V=800.0 PL=0
MOVL C01818 V=800.0 PL=0
MOVL C01819 V=800.0 PL=0
MOVL C01820 V=800.0 PL=0
MOVL C01821 V=800.0 PL=0
MOVL C01822 V=800.0 PL=0
MOVL C01823 V=800.0 PL=0
MOVL C01824 V=800.0 PL=0
MOVL C01825 V=800.0 PL=0
MOVL C01826 V=800.0 PL=0
MOVL C01827 V=800.0 PL=0
MOVL C01828 V=800.0 PL=0
MOVL C01829 V=800.0 PL=0
MOVL C01830 V=800.0 PL=0
MOVL C01831 V=800.0 PL=0
MOVL C01832 V=800.0 PL=0
MOVL C01833 V=800.0 PL=0
MOVL C01834 V=800.0 PL=0
MOVL C01835 V=800.0 PL=0
MOVL C01836 V=800.0 PL=0
MOVL C01837 V=800.0 PL=0
MOVL C01838 V=800.0 PL=0
MOVL C01839 V=800.0 PL=0
MOVL C01840 V=800.0 PL=0
MOVL C01841 V=800.0 PL=0
MOVL C01842 V=800.0 PL=0
MOVL C01843 V=800.0 PL=0
MOVL C01844 V=800.0 PL=0
MOVL C01845 V=800.0 PL=0
MOVL C01846 V=800.0 PL=0
MOVL C01847 V=800.0 PL=0
MOVL C01848 V=800.0 PL=0
MOVL C01849 V=800.0 PL=0
MOVL C01850 V=800.0 PL=0
MOVL C01851 V=800.0 PL=0
MOVL C01852 V=800.0 PL=0
MOVL C01853 V=800.0 PL=0
MOVL C01854 V=800.0 PL=0
MOVL C01855 V=800.0 PL=0
MOVL C01856 V=800.0 PL=0
MOVL C01857 V=800.0 PL=0
MOVL C01858 V=800.0 PL=0
MOVL C01859 V=800.0 PL=0
MOVL C01860 V=800.0 PL=0
MOVL C01861 V=800.0 PL=0
MOVL C01862 V=800.0 PL=0
MOVL C01863 V=800.0 PL=0
MOVL C01864 V=800.0 PL=0
MOVL C01865 V=800.0 PL=0
MOVL C01866 V=800.0 PL=0
MOVL C01867 V=800.0 PL=0
MOVL C01868 V=800.0 PL=0
MOVL C01869 V=800.0 PL=0
MOVL C01870 V=800.0 PL=0
MOVL C01871 V=800.0 PL=0
MOVL C01872 V=800.0 PL=0
MOVL C01873 V=800.0 PL=0
MOVL C01874 V=800.0 PL=0
MOVL C01875 V=800.0 PL=0
MOVL C01876 V=800.0 PL=0
MOVL C01877 V=800.0 PL=0
MOVL C01878 V=800.0 PL=0
MOVL C01879 V=800.0 PL=0
MOVL C01880 V=800.0 PL=0
MOVL C01881 V=800.0 PL=0
MOVL C01882 V=800.0 PL=0
MOVL C01883 V=800.0 PL=0
MOVL C01884 V=800.0 PL=0
MOVL C01885 V=800.0 PL=0
MOVL C01886 V=800.0 PL=0
MOVL C01887 V=800.0 PL=0
MOVL C01888 V=800.0 PL=0
MOVL C01889 V=800.0 PL=0
MOVL C01890 V=800.0 PL=0
MOVL C01891 V=800.0 PL=0
MOVL C01892 V=800.0 PL=0
MOVL C01893 V=800.0 PL=0
MOVL C01894 V=800.0 PL=0
MOVL C01895 V=800.0 PL=0
MOVL C01896 V=800.0 PL=0
MOVL C01897 V=800.0 PL=0
MOVL C01898 V=800.0 PL=0
MOVL C01899 V=800.0 PL=0
MOVL C01900 V=800.0 PL=0
MOVL C01901 V=800.0 PL=0
MOVL C01902 V=800.0 PL=0
MOVL C01903 V=800.0 PL=0
MOVL C01904 V=800.0 PL=0
MOVL C01905 V=800.0 PL=0
MOVL C01906 V=800.0 PL=0
MOVL C01907 V=800.0 PL=0
MOVL C01908 V=800.0 PL=0
MOVL C01909 V=800.0 PL=0
MOVL C01910 V=800.0 PL=0
MOVL C01911 V=800.0 PL=0
MOVL C01912 V=800.0 PL=0
MOVL C01913 V=800.0 PL=0
MOVL C01914 V=800.0 PL=0
MOVL C01915 V=800.0 PL=0
MOVL C01916 V=800.0 PL=0
MOVL C01917 V=800.0 PL=0
MOVL C01918 V=800.0 PL=0
MOVL C01919 V=800.0 PL=0
MOVL C01920 V=800.0 PL=0
MOVL C01921 V=800.0 PL=0
MOVL C01922 V=800.0 PL=0
MOVL C01923 V=800.0 PL=0
MOVL C01924 V=800.0 PL=0
MOVL C01925 V=800.0 PL=0
MOVL C01926 V=800.0 PL=0
MOVL C01927 V=800.0 PL=0
MOVL C01928 V=800.0 PL=0
MOVL C01929 V=800.0 PL=0
MOVL C01930 V=800.0 PL=0
MOVL C01931 V=800.0 PL=0
MOVL C01932 V=800.0 PL=0
MOVL C01933 V=800.0 PL=0
MOVL C01934 V=800.0 PL=0
MOVL C01935 V=800.0 PL=0
MOVL C01936 V=800.0 PL=0
MOVL C01937 V=800.0 PL=0
MOVL C01938 V=800.0 PL=0
MOVL C01939 V=800.0 PL=0
MOVL C01940 V=800.0 PL=0
MOVL C01941 V=800.0 PL=0
MOVL C01942 V=800.0 PL=0
MOVL C01943 V=800.0 PL=0
MOVL C01944 V=800.0 PL=0
MOVL C01945 V=800.0 PL=0
MOVL C01946 V=800.0 PL=0
MOVL C01947 V=800.0 PL=0
MOVL C01948 V=800.0 PL=0
MOVL C01949 V=800.0 PL=0
MOVL C01950 V=800.0 PL=0
MOVL C01951 V=800.0 PL=0
MOVL C01952 V=800.0 PL=0
MOVL C01953 V=800.0 PL=0
MOVL C01954 V=800.0 PL=0
MOVL C01955 V=800.0 PL=0
MOVL C01956 V=800.0 PL=0
MOVL C01957 V=800.0 PL=0
MOVL C01958 V=800.0 PL=0
MOVL C01959 V=800.0 PL=0
MOVL C01960 V=800.0 PL=0
MOVL C01961 V=800.0 PL=0
MOVL C01962 V=800.0 PL=0
MOVL C01963 V=800.0 PL=0
MOVL C01964 V=800.0 PL=0
MOVL C01965 V=800.0 PL=0
MOVL C01966 V=800.0 PL=0
MOVL C01967 V=800.0 PL=0
MOVL C01968 V=800.0 PL=0
MOVL C01969 V=800.0 PL=0
MOVL C01970 V=800.0 PL=0
MOVL C01971 V=800.0 PL=0
MOVL C01972 V=800.0 PL=0
MOVL C01973 V=800.0 PL=0
MOVL C01974 V=800.0 PL=0
MOVL C01975 V=800.0 PL=0
MOVL C01976 V=800.0 PL=0
MOVL C01977 V=800.0 PL=0
MOVL C01978 V=800.0 PL=0
MOVL C01979 V=800.0 PL=0
MOVL C01980 V=800.0 PL=0
MOVL C01981 V=800.0 PL=0
MOVL C01982 V=800.0 PL=0
MOVL C01983 V=800.0 PL=0
MOVL C01984 V=800.0 PL=0
MOVL C01985 V=800.0 PL=0
MOVL C01986 V=800.0 PL=0
MOVL C01987 V=800.0 PL=0
MOVL C01988 V=800.0 PL=0
MOVL C01989 V=800.0 PL=0
MOVL C01990 V=800.0 PL=0
MOVL C01991 V=800.0 PL=0
MOVL C01992 V=800.0 PL=0
MOVL C01993 V=800.0 PL=0
MOVL C01994 V=800.0 PL=0
MOVL C01995 V=800.0 PL=0
MOVL C01996 V=800.0 PL=0
MOVL C01997 V=800.0 PL=0
MOVL C01998 V=800.0 PL=0
MOVL C01999 V=800.0 PL=0
MOVL C02000 V=800.0 PL=0
MOVL C02001 V=800.0 PL=0
